DATA_BLOCK "pressure"   // DB71
{ S7_Optimized_Access := 'TRUE' }
VERSION : 0.1
// stored: AutoNumber true, DBAccessibleFromOPCUA true, IsOnlyStoredInLoadMemory false, IsRetainMemResEnabled false, IsWriteProtectedInAS false, MemoryReserve 100
   VAR RETAIN
      "A" : Struct
         "pressure at 20mA" : Real := 160.0;
         "Maximum Pressure user" : Real := 10.0;
         "maximum pressure Admin" : Real := 10.0;
         "minimum Pressure" : Real := 1.5;
      END_STRUCT;
      "B" : Struct
         "pressure at 20mA" : Real := 160.0;
         "Maximum Pressure user" : Real := 10.0;
         "maximum pressure Admin" : Real := 10.0;
         "minimum Pressure" : Real := 1.5;
      END_STRUCT;
   END_VAR
   VAR
      "Control A" : Struct
         "Over pressure occured" : Bool := FALSE;
         "under pressure Occured" : Bool := FALSE;
      END_STRUCT;
      "Control B" : Struct
         "Over pressure occured" : Bool := FALSE;
         "under pressure Occured" : Bool := FALSE;
      END_STRUCT;
      "pump A Inlet" : Real := 1.50463;
      "pump B Inlet" : Real := 1.545139;
      "pump A Outlet" : Real := 0.1808449;
      "pump B Outlet" : Real := 0.1139323;
      "Vessel A1 mbar" : DInt := 0;
      "Vessel A2 mbar" : DInt := 0;
      "Vessel B2 mbar" : DInt := 0;
      "Vessel B1 mbar" : DInt := 0;
   END_VAR
   VAR RETAIN
      "Over pressure Delay time user" : DInt := 1000;
      "over pressure delay time admin" : DInt := 10000;
      "under pressure delay time" : DInt := 1000;
      "Vaccum  sensor range" : Struct
         A1mbar : DInt := 9000;
         A2mbar : DInt := 9000;
         B1mbar : DInt := 9000;
         B2mbar : DInt := 9000;
         A1bar : Real := 9.0;
         A2bar : Real := 9.0;
         B1bar : Real := 9.0;
         B2bar : Real := 0.0;
      END_STRUCT;
   END_VAR
   VAR
      "vessel A1 bar" : Real := 0.0;
      "vessel A2 bar" : Real := 0.0;
      "vessel B1 bar" : Real := 0.0;
      "vessel B2 bar" : Real := 0.0;
      Misc : Struct
         "Pump A normx valueIN" : Real := 0.009403936;
         "Pump B normx valueIN" : Real := 0.009657118;
         "Pump A Scalx valueIN" : Real := 1.50463;
         "Pump B Scalx valueIN" : Real := 1.545139;
         "Pump A normx valueOUT" : Real := 0.007233796;
         "Pump B normx valueOUT" : Real := 0.004557292;
         "Pump A Scalx valueOUT" : Real := 0.1808449;
         "Pump B Scalx valueOUT" : Real := 0.1139323;
         "normx Tank A1" : Real := 0.0;
         "normx Tank A2" : Real := 0.0;
         "normx Tank B1" : Real := 0.0;
         "normx Tank B2" : Real := 0.0;
         "scalx Tank A1" : Real := 0.0;
         "scalx Tank A2" : Real := 0.0;
         "scalx Tank B1" : Real := 0.0;
         "scalx Tank B2" : Real := 0.0;
      END_STRUCT;
      "Control Vessel A1" : Struct
         "under pressure" : Bool := FALSE;
         "Over pressure open release valve" : Bool := FALSE;
      END_STRUCT;
      "Control Vessel A2" : Struct
         "under pressure" : Bool := FALSE;
         "Over pressure open release valve" : Bool := FALSE;
      END_STRUCT;
      "Control Vessel B1" : Struct
         "under pressure" : Bool := FALSE;
         "Over pressure open release valve" : Bool := FALSE;
      END_STRUCT;
      "Control Vessel B2" : Struct
         "under pressure" : Bool := FALSE;
         "Over pressure open release valve" : Bool := FALSE;
      END_STRUCT;
   END_VAR
   VAR RETAIN
      A_Outlet : Struct
         "pressure at 20mA" : Real := 25.0;
         "Maximum Pressure user" : Real := 20.0;
         "maximum pressure Admin" : Real := 20.0;
         "minimum Pressure" : Real := 1.0;
      END_STRUCT;
      B_Outlet : Struct
         "pressure at 20mA" : Real := 25.0;
         "Maximum Pressure user" : Real := 20.0;
         "maximum pressure Admin" : Real := 20.0;
         "minimum Pressure" : Real := 1.0;
      END_STRUCT;
   END_VAR
   VAR
      "Control A_Outlet" : Struct
         "Over pressure occured" : Bool := FALSE;
         "under pressure Occured" : Bool := FALSE;
      END_STRUCT;
      "Control B_Outlet" : Struct
         "Over pressure occured" : Bool := FALSE;
         "under pressure Occured" : Bool := FALSE;
      END_STRUCT;
   END_VAR
   VAR RETAIN
      Outlet_PT_ENABLE : Bool := TRUE;
   END_VAR
BEGIN
END_DATA_BLOCK

DATA_BLOCK "vessel"   // DB75
{ S7_Optimized_Access := 'TRUE' }
VERSION : 0.1
// stored: AutoNumber true, DBAccessibleFromOPCUA true, IsOnlyStoredInLoadMemory false, IsRetainMemResEnabled false, IsWriteProtectedInAS false, MemoryReserve 100
   VAR RETAIN
      "Duration pressure equalization" : Struct
         "A" : Int := 10;
         "B" : Int := 10;
      END_STRUCT;
      "amibient pressure" : Int := 900;
      "hysteresis ambient pressure" : Int := 50;
      "working pressure" : Struct
         "A" : Real := 3.0;
         "A+" : Real;
         "A-" : Real;
         "B" : Real := 3.0;
         "B+" : Real;
         "B-" : Real;
      END_STRUCT;
      "working pressure hysteresis" : Struct
         "A" : Real;
         "B" : Real;
      END_STRUCT;
   END_VAR
   VAR
      "Vaccum sensor selection" : Struct
         "selection A" : Int;
         "selection B" : Int;
         "A selected" : Bool;
         "B selected" : Bool;
         "A or B selected" : Bool;
      END_STRUCT;
      "Evacuation set Vaccum" : Struct
         A1 : Int;
         A2 : Int;
         B1 : Int;
         B2 : Int;
      END_STRUCT;
      "Evacuation Real vaccum" : Struct
         A1 : Int;
         A2 : Int;
         B1 : Int;
         B2 : Int;
      END_STRUCT;
      "Evacuation Time set" : Struct
         A1 : Int;
         A2 : Int;
         B1 : Int;
         B2 : Int;
      END_STRUCT;
      "Evacuation Time Real" : Struct
         A1 : Int;
         A2 : Int;
         B1 : Int;
         B2 : Int;
      END_STRUCT;
   END_VAR
   VAR RETAIN
      "preparation status" : Struct
         A1 : Int;
         A2 : Int;
         B1 : Int;
         B2 : Int;
      END_STRUCT;
      "monitor status" : Struct
         A1 : Int;
         A2 : Int;
         B1 : Int;
         B2 : Int;
      END_STRUCT;
      "Activate vessel" : Struct
         A1 : Bool;
         A2 : Bool;
         B1 : Bool;
         B2 : Bool;
      END_STRUCT;
   END_VAR
   VAR
      "A status" : Int;
      "B status" : Int;
   END_VAR
BEGIN
END_DATA_BLOCK

DATA_BLOCK "vessel_1"   // DB81
{ S7_Optimized_Access := 'TRUE' }
VERSION : 0.1
// stored: AutoNumber true, DBAccessibleFromOPCUA true, IsOnlyStoredInLoadMemory false, IsRetainMemResEnabled false, IsWriteProtectedInAS false, MemoryReserve 100
   VAR RETAIN
      "Duration pressure equalization" : Struct
         "A" : Int;
         "B" : Int;
      END_STRUCT;
      "amibient pressure" : Int;
      "hysteresis ambient pressure" : Int;
      "working pressure" : Struct
         "A" : Real;
         "A+" : Real;
         "A-" : Real;
         "B" : Real;
         "B+" : Real;
         "B-" : Real;
      END_STRUCT;
      "working pressure hysteresis" : Struct
         "A" : Real;
         "B" : Real;
      END_STRUCT;
   END_VAR
   VAR
      "Vaccum sensor selection" : Struct
         "selection A" : Int;
         "selection B" : Int;
         "A selected" : Bool;
         "B selected" : Bool;
         "A or B selected" : Bool;
      END_STRUCT;
      "Ready status" : Struct
         A1 : Int;
         A2 : Int;
         B1 : Int;
      END_STRUCT;
      "Evacuation set Vaccum" : Struct
         A1 : Int;
         A2 : Int;
         B1 : Int;
      END_STRUCT;
      "Evacuation Real vaccum" : Struct
         A1 : Int;
         A2 : Int;
         B1 : Int;
      END_STRUCT;
      "Evacuation Time set" : Struct
         A1 : Int;
         A2 : Int;
         B1 : Int;
      END_STRUCT;
      "Evacuation Time Real" : Struct
         A1 : Int;
         A2 : Int;
         B1 : Int;
      END_STRUCT;
   END_VAR
   VAR RETAIN
      "Active vessel" : Struct
         A1 : Bool;
         A2 : Bool;
         "A" : Bool;
         B1 : Bool;
      END_STRUCT;
      "preparation status" : Struct
         A1 : Int;
         A2 : Int;
         B1 : Int;
      END_STRUCT;
      "monitor status" : Struct
         "A" : Int;
         "B" : Int;
         C : Int;
      END_STRUCT;
      "Activate vessel" : Struct
         A1 : Bool;
         A2 : Bool;
         B1 : Bool;
      END_STRUCT;
   END_VAR
   VAR
      Ready : Struct
         A1 : Bool;
         A2 : Bool;
         B1 : Bool;
      END_STRUCT;
      "Activate vessel HMI" : Struct
         A1 : Bool;
         A2 : Bool;
         B1 : Bool;
      END_STRUCT;
      "DeActivate vessel HMI" : Struct
         A1 : Bool;
         A2 : Bool;
         B1 : Bool;
      END_STRUCT;
   END_VAR
BEGIN
END_DATA_BLOCK

DATA_BLOCK "Alarm_DB"   // DB36
{ S7_Optimized_Access := 'FALSE' }
VERSION : 0.1
// stored: AutoNumber true, DBAccessibleFromOPCUA true, IsOnlyStoredInLoadMemory false, IsWriteProtectedInAS false
   VAR
      input : Struct
         alarm : Array[0..95] of Bool;   // Connect the alarm inputs according to the alarm list
         ack : Array[0..95] of Bool;
      END_STRUCT;
      output : Struct
         alarm_reg : Array[0..95] of Bool;
      END_STRUCT;
      i : Int;
      alarmhmi : Bool;
      alarmRegister1 : Word;
      alarmRegister2 : Word;
      alarmRegister3 : Word;
      alarmRegister4 : Word;
      alarmRegister5 : Word;
      reset : Array[0..95] of Bool;
   END_VAR
BEGIN
   // input.alarm[0] : reg1 bit 8
   // input.alarm[1] : reg1 bit 9
   // input.alarm[2] : reg1 bit 10
   // input.alarm[3] : reg1 bit 11
   // input.alarm[4] : reg1 bit 12
   // input.alarm[5] : reg1 bit 13
   // input.alarm[6] : reg1 bit 14
   // input.alarm[7] : reg1 bit 15
   // input.alarm[8] : reg1 bit 0
   // input.alarm[9] : reg1 bit 1
   // input.alarm[10] : reg1 bit 2
   // input.alarm[11] : reg1 bit 3
   // input.alarm[12] : reg1 bit 4
   // input.alarm[13] : reg1 bit 5
   // input.alarm[14] : reg1 bit 6
   // input.alarm[15] : reg1 bit 0
   // input.alarm[16] : reg2 bit 8
   // input.alarm[17] : reg2 bit 9
   // input.alarm[18] : reg2 bit 10
   // input.alarm[19] : reg2 bit 11
   // input.alarm[20] : reg2 bit 12
   // input.alarm[21] : reg2 bit 13
   // input.alarm[22] : reg2 bit 14
   // input.alarm[23] : reg2 bit 15
   // input.alarm[24] : reg2 bit 7
   // input.alarm[25] : reg2 bit 6
   // input.alarm[26] : reg2 bit 5
   // input.alarm[27] : reg2 bit 4
   // input.alarm[28] : reg2 bit 3
   // input.alarm[29] : reg2 bit 2
   // input.alarm[30] : reg2 bit 1
   // input.alarm[31] : reg2 bit 0
   // input.alarm[32] : reg3 bit 8
   // input.alarm[33] : reg3 bit 9
   // input.alarm[34] : reg3 bit 10
   // input.alarm[35] : reg3 bit 11
   // input.alarm[36] : reg3 bit 12
   // input.alarm[37] : reg3 bit 13
   // input.alarm[38] : reg3 bit 14
   // input.alarm[39] : reg3 bit 15
   // input.alarm[40] : reg3 bit 7
   // input.alarm[41] : reg3 bit 6
   // input.alarm[42] : reg3 bit 5
   // input.alarm[43] : reg3 bit 4
   // input.alarm[44] : reg3 bit 3
   // input.alarm[45] : reg3 bit 2
   // input.alarm[46] : reg3 bit 1
   // input.alarm[47] : reg3 bit 0
   // input.alarm[48] : reg4 bit 8
   // input.alarm[49] : reg4 bit 9
   // input.alarm[50] : reg4 bit 10
   // input.alarm[51] : reg4 bit 11
   // input.alarm[52] : reg4 bit 12
   // input.alarm[53] : reg4 bit 13
   // input.alarm[54] : reg4 bit 14
   // input.alarm[55] : reg4 bit 15
   // input.alarm[56] : reg4 bit 7
   // input.alarm[57] : reg4 bit 6
   // input.alarm[58] : reg4 bit 5
   // input.alarm[59] : reg4 bit 4
   // input.alarm[60] : reg4 bit 3
   // input.alarm[61] : reg4 bit 2
   // input.alarm[62] : reg4 bit 1
   // input.alarm[63] : reg4 bit 0
   // input.alarm[64] : reg5 bit 8
   // input.alarm[65] : reg5 bit 9
   // input.alarm[66] : reg5 bit 10
   // input.alarm[67] : reg5 bit 11
   // input.alarm[68] : reg5 bit 12
   // input.alarm[69] : reg5 bit 13
   // input.alarm[70] : reg5 bit 14
   // input.alarm[71] : reg5 bit 15
   // input.alarm[72] : reg5 bit 7
   // input.alarm[73] : reg5 bit 6
   // input.alarm[74] : reg5 bit 5
   // input.alarm[75] : reg5 bit 4
   // input.alarm[76] : reg5 bit 3
   // input.alarm[77] : reg5 bit 2
   // input.alarm[78] : reg5 bit 1
   // input.alarm[79] : reg5 bit 0
END_DATA_BLOCK

DATA_BLOCK "Heater settings"   // DB138
{ S7_Optimized_Access := 'TRUE' }
VERSION : 0.1
// stored: AutoNumber true, DBAccessibleFromOPCUA true, IsOnlyStoredInLoadMemory false, IsRetainMemResEnabled false, IsWriteProtectedInAS false, MemoryReserve 100
   VAR RETAIN
      "Heater 1" : Struct
         "set temperature" : Real;
         "preshutdown temperature" : Real;
         "Limit under temparature" : Real;
         "Limit Over temperature" : Real;
         "Heating adjustment hysteresis" : Real;
         "Minimum ON time" : Real;
         "Minimum Off time" : Real;
      END_STRUCT;
      "Heater 2" : Struct
         "set temperature" : Real;
         "preshutdown temperature" : Real;
         "Limit under temparature" : Real;
         "Limit Over temperature" : Real;
         "Heating adjustment hysteresis" : Real;
         "Minimum ON time" : Real;
         "Minimum Off time" : Real;
      END_STRUCT;
      "Heater 3" : Struct
         "set temperature" : Real;
         "preshutdown temperature" : Real;
         "Limit under temparature" : Real;
         "Limit Over temperature" : Real;
         "Heating adjustment hysteresis" : Real;
         "Minimum ON time" : Real;
         "Minimum Off time" : Real;
      END_STRUCT;
      "Heater 4" : Struct
         "set temperature" : Real;
         "preshutdown temperature" : Real;
         "Limit under temparature" : Real;
         "Limit Over temperature" : Real;
         "Heating adjustment hysteresis" : Real;
         "Minimum ON time" : Real;
         "Minimum Off time" : Real;
      END_STRUCT;
      "heater EN 1" : Bool;
      "heater EN 2" : Bool;
      "heater EN 3" : Bool;
      "heater EN 4" : Bool;
   END_VAR
BEGIN
END_DATA_BLOCK

DATA_BLOCK "Heatercontrol"   // DB140
{ S7_Optimized_Access := 'TRUE' }
VERSION : 0.1
// stored: AutoNumber true, DBAccessibleFromOPCUA true, IsOnlyStoredInLoadMemory false, IsRetainMemResEnabled false, IsWriteProtectedInAS false, MemoryReserve 100
   VAR RETAIN
      ON : Struct
         heater1 : Bool;
         heater2 : Bool;
         heater3 : Bool;
         heater4 : Bool;
      END_STRUCT;
      "heater ON HMI" : Bool;
   END_VAR
   VAR
      "Show heater Button" : Bool;
   END_VAR
BEGIN
END_DATA_BLOCK

DATA_BLOCK "heater status"   // DB141
{ S7_Optimized_Access := 'TRUE' }
VERSION : 0.1
// stored: AutoNumber true, DBAccessibleFromOPCUA true, IsOnlyStoredInLoadMemory false, IsRetainMemResEnabled false, IsWriteProtectedInAS false, MemoryReserve 100
   VAR
      temperature : Struct
         heater1 : Real;
         heater2 : Real;
         heater3 : Real;
         heater4 : Real;
      END_STRUCT;
   END_VAR
   VAR RETAIN
      "p100 connection okay" : Struct
         heater1 : Bool;
         heater2 : Bool;
         heater3 : Bool;
         heater4 : Bool;
      END_STRUCT;
   END_VAR
   VAR
      "Limit under temperature" : Struct
         heater1 : Bool;
         heater2 : Bool;
         heater3 : Bool;
         heater4 : Bool;
      END_STRUCT;
      "Limit Over temperature" : Struct
         heater1 : Bool;
         heater2 : Bool;
         heater3 : Bool;
         heater4 : Bool;
      END_STRUCT;
      "Dispensing Stop under temperature heater" { ExternalAccessible := 'False'; ExternalVisible := 'False'; ExternalWritable := 'False'} : Array[1..4] of Bool;
      "Critical Fault Stop Dispense Temperature NOK" : Bool;
      heater_nok : Bool;
   END_VAR
BEGIN
END_DATA_BLOCK

DATA_BLOCK "selection_machie_db"   // DB18
{ S7_Optimized_Access := 'TRUE' }
VERSION : 0.1
// stored: AutoNumber true, DBAccessibleFromOPCUA true, IsOnlyStoredInLoadMemory false, IsRetainMemResEnabled false, IsWriteProtectedInAS false, MemoryReserve 100
   VAR
      "1k_2k" : Bool;
   END_VAR
BEGIN
END_DATA_BLOCK

ORGANIZATION_BLOCK "Main"   // OB1, LAD, ProgramCycle
TITLE = "Main Program Sweep (Cycle)"
{ S7_Optimized_Access := 'TRUE' }
VERSION : 0.1
// stored: AutoNumber true, IsIECCheckEnabled false, SetENOAutomatically false
   VAR_INPUT
      Initial_Call : Bool;   // Initial call of this OB
      Remanence : Bool;   // =True, if remanent data are available
   END_VAR
   VAR_TEMP
      temp1 : Bool;
      temp2 : Bool;
      temp3 : Bool;
      temp4 : Bool;
   END_VAR
   VAR_TEMP   // added for the SCL form of the ladder/FBD networks
      _w1 : Bool;
      _w2 : Bool;
      _w3 : Bool;
      _w4 : Bool;
      _w5 : Bool;
      _w6 : Bool;
      _w7 : Bool;
      _w8 : Bool;
      _w9 : Bool;
      _w10 : Bool;
      _w11 : Bool;
      _w12 : Bool;
      _w13 : Bool;
      _w14 : Bool;
      _w15 : Bool;
      _w16 : Bool;
   END_VAR
BEGIN

REGION Network 1: SFC1
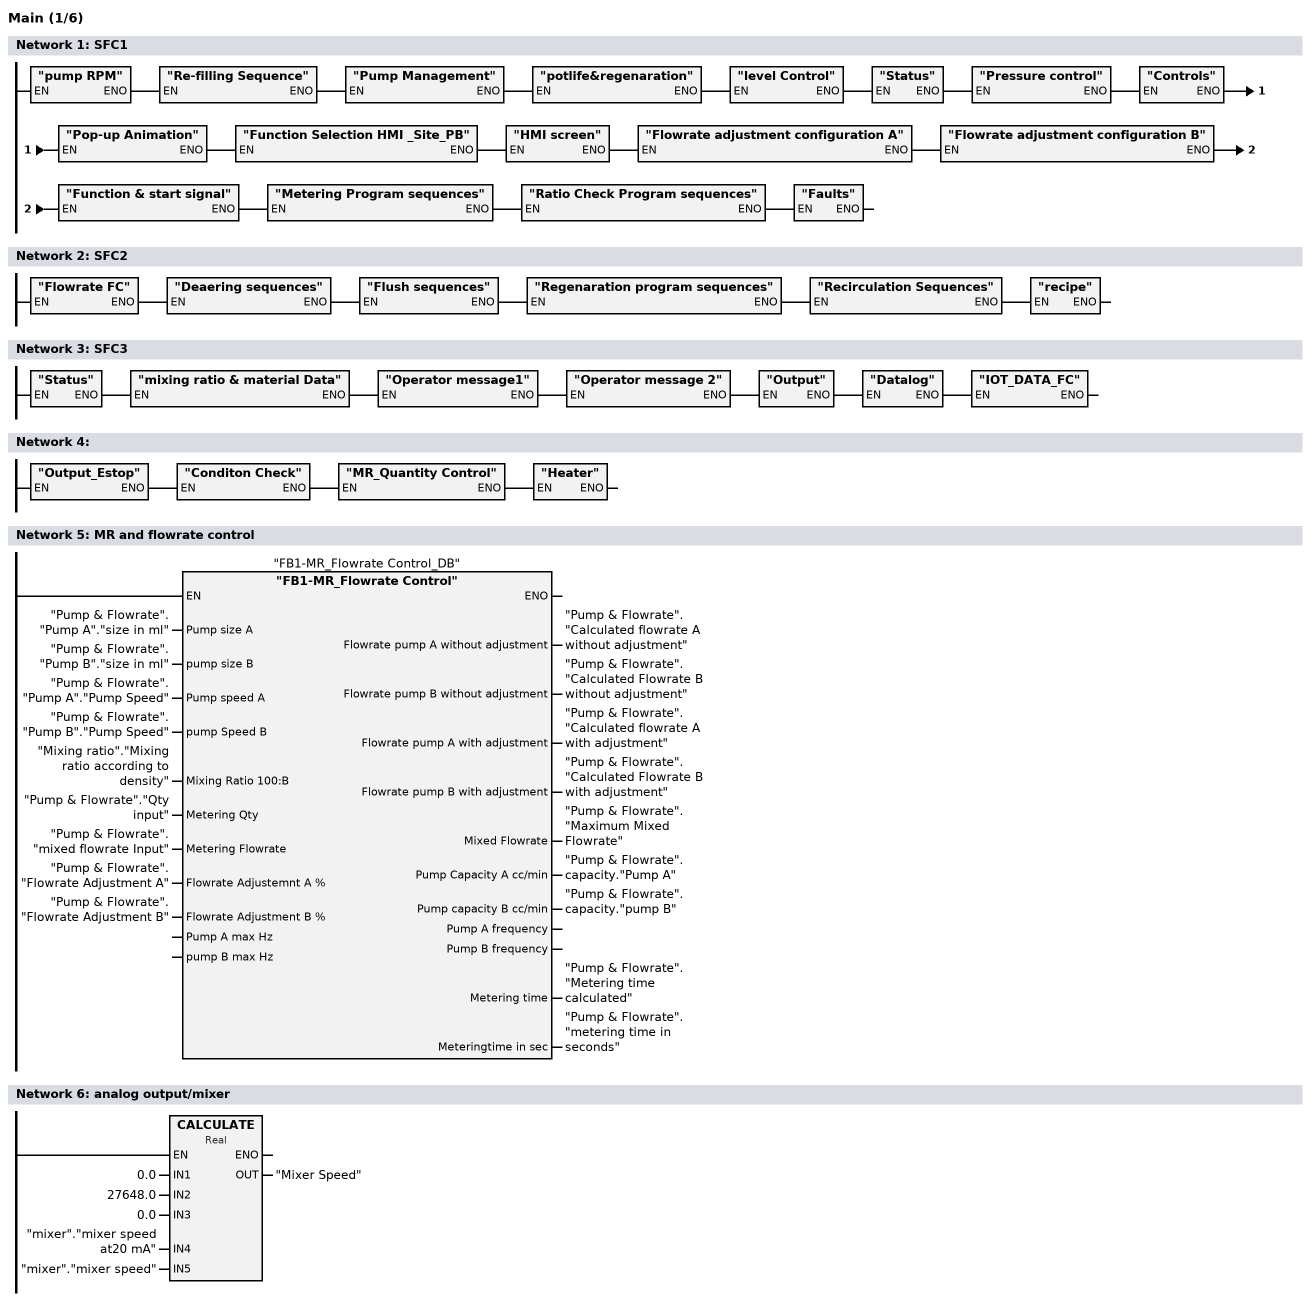
   RUNG wire#powerrail
      "pump RPM"()
      "Re-filling Sequence"()
      "Pump Management"()
      "potlife&regenaration"()
      "level Control"()
      "Status"()
      "Pressure control"()
      "Controls"()
      "Pop-up Animation"()
      "Function Selection HMI _Site_PB"()
      "HMI screen"()
      "Flowrate adjustment configuration A"()
      "Flowrate adjustment configuration B"()
      "Function & start signal"()
      "Metering Program sequences"()
      "Ratio Check Program sequences"()
      "Faults"()
   END_RUNG
   // the same network as SCL:
   "pump RPM"(ENO => #_w1);
   "Re-filling Sequence"(EN := #_w1, ENO => #_w2);
   "Pump Management"(EN := #_w2, ENO => #_w3);
   "potlife&regenaration"(EN := #_w3, ENO => #_w4);
   "level Control"(EN := #_w4, ENO => #_w5);
   "Status"(EN := #_w5, ENO => #_w6);
   "Pressure control"(EN := #_w6, ENO => #_w7);
   "Controls"(EN := #_w7, ENO => #_w8);
   "Pop-up Animation"(EN := #_w8, ENO => #_w9);
   "Function Selection HMI _Site_PB"(EN := #_w9, ENO => #_w10);
   "HMI screen"(EN := #_w10, ENO => #_w11);
   "Flowrate adjustment configuration A"(EN := #_w11, ENO => #_w12);
   "Flowrate adjustment configuration B"(EN := #_w12, ENO => #_w13);
   "Function & start signal"(EN := #_w13, ENO => #_w14);
   "Metering Program sequences"(EN := #_w14, ENO => #_w15);
   "Ratio Check Program sequences"(EN := #_w15, ENO => #_w16);
   IF #_w16 THEN "Faults"(); END_IF;
END_REGION

REGION Network 2: SFC2
   RUNG wire#powerrail
      "Flowrate FC"()
      "Deaering sequences"()
      "Flush sequences"()
      "Regenaration program sequences"()
      "Recirculation Sequences"()
      "recipe"()
   END_RUNG
   // the same network as SCL:
   "Flowrate FC"(ENO => #_w1);
   "Deaering sequences"(EN := #_w1, ENO => #_w2);
   "Flush sequences"(EN := #_w2, ENO => #_w3);
   "Regenaration program sequences"(EN := #_w3, ENO => #_w4);
   "Recirculation Sequences"(EN := #_w4, ENO => #_w5);
   IF #_w5 THEN "recipe"(); END_IF;
END_REGION

REGION Network 3: SFC3
   RUNG wire#powerrail
      "Status"()
      "mixing ratio & material Data"()
      "Operator message1"()
      "Operator message 2"()
      "Output"()
      "Datalog"()
      "IOT_DATA_FC"()
   END_RUNG
   // the same network as SCL:
   "Status"(ENO => #_w1);
   "mixing ratio & material Data"(EN := #_w1, ENO => #_w2);
   "Operator message1"(EN := #_w2, ENO => #_w3);
   "Operator message 2"(EN := #_w3, ENO => #_w4);
   "Output"(EN := #_w4, ENO => #_w5);
   "Datalog"(EN := #_w5, ENO => #_w6);
   IF #_w6 THEN "IOT_DATA_FC"(); END_IF;
END_REGION

REGION Network 4
   RUNG wire#powerrail
      "Output_Estop"()
      "Conditon Check"()
      "MR_Quantity Control"()
      "Heater"()
   END_RUNG
   // the same network as SCL:
   "Output_Estop"(ENO => #_w1);
   "Conditon Check"(EN := #_w1, ENO => #_w2);
   "MR_Quantity Control"(EN := #_w2, ENO => #_w3);
   IF #_w3 THEN "Heater"(); END_IF;
END_REGION

REGION Network 5: MR and flowrate control
   "FB1-MR_Flowrate Control_DB"("Pump size A" := "Pump & Flowrate"."Pump A"."size in ml",   // "FB1-MR_Flowrate Control"
                           "pump size B" := "Pump & Flowrate"."Pump B"."size in ml",
                           "Pump speed A" := "Pump & Flowrate"."Pump A"."Pump Speed",
                           "pump Speed B" := "Pump & Flowrate"."Pump B"."Pump Speed",
                           "Mixing Ratio 100:B" := "Mixing ratio"."Mixing ratio according to density",
                           "Metering Qty" := "Pump & Flowrate"."Qty input",
                           "Metering Flowrate" := "Pump & Flowrate"."mixed flowrate Input",
                           "Flowrate Adjustemnt A %" := "Pump & Flowrate"."Flowrate Adjustment A",
                           "Flowrate Adjustment B %" := "Pump & Flowrate"."Flowrate Adjustment B",
                           "Flowrate pump A without adjustment" => "Pump & Flowrate"."Calculated flowrate A without adjustment",
                           "Flowrate pump B without adjustment" => "Pump & Flowrate"."Calculated Flowrate B without adjustment",
                           "Flowrate pump A with adjustment" => "Pump & Flowrate"."Calculated flowrate A with adjustment",
                           "Flowrate pump B with adjustment" => "Pump & Flowrate"."Calculated Flowrate B  with adjustment",
                           "Mixed Flowrate" => "Pump & Flowrate"."Maximum Mixed Flowrate",
                           "Pump Capacity A cc/min" => "Pump & Flowrate".capacity."Pump A",
                           "Pump capacity B cc/min" => "Pump & Flowrate".capacity."pump B",
                           "Metering time" => "Pump & Flowrate"."Metering time calculated",
                           "Meteringtime in sec" => "Pump & Flowrate"."metering time in seconds");
END_REGION

REGION Network 6: analog output/mixer
   RUNG wire#powerrail
      { S7_Templates := "SrcType := Real"; S7_Expression := "(IN2-IN1)*(IN5-IN3)/(IN4-IN3)+IN1" } Calculate(in1 := 0.0, in2 := 27648.0, in3 := 0.0, in4 := "mixer"."mixer speed at20 mA", in5 := "mixer"."mixer speed", out => "Mixer Speed")
   END_RUNG
   // the same network as SCL:
   "Mixer Speed" := (27648.0-0.0)*("mixer"."mixer speed"-0.0)/("mixer"."mixer speed at20 mA"-0.0)+0.0;
END_REGION

REGION Network 7: Pump A Analog output without PID
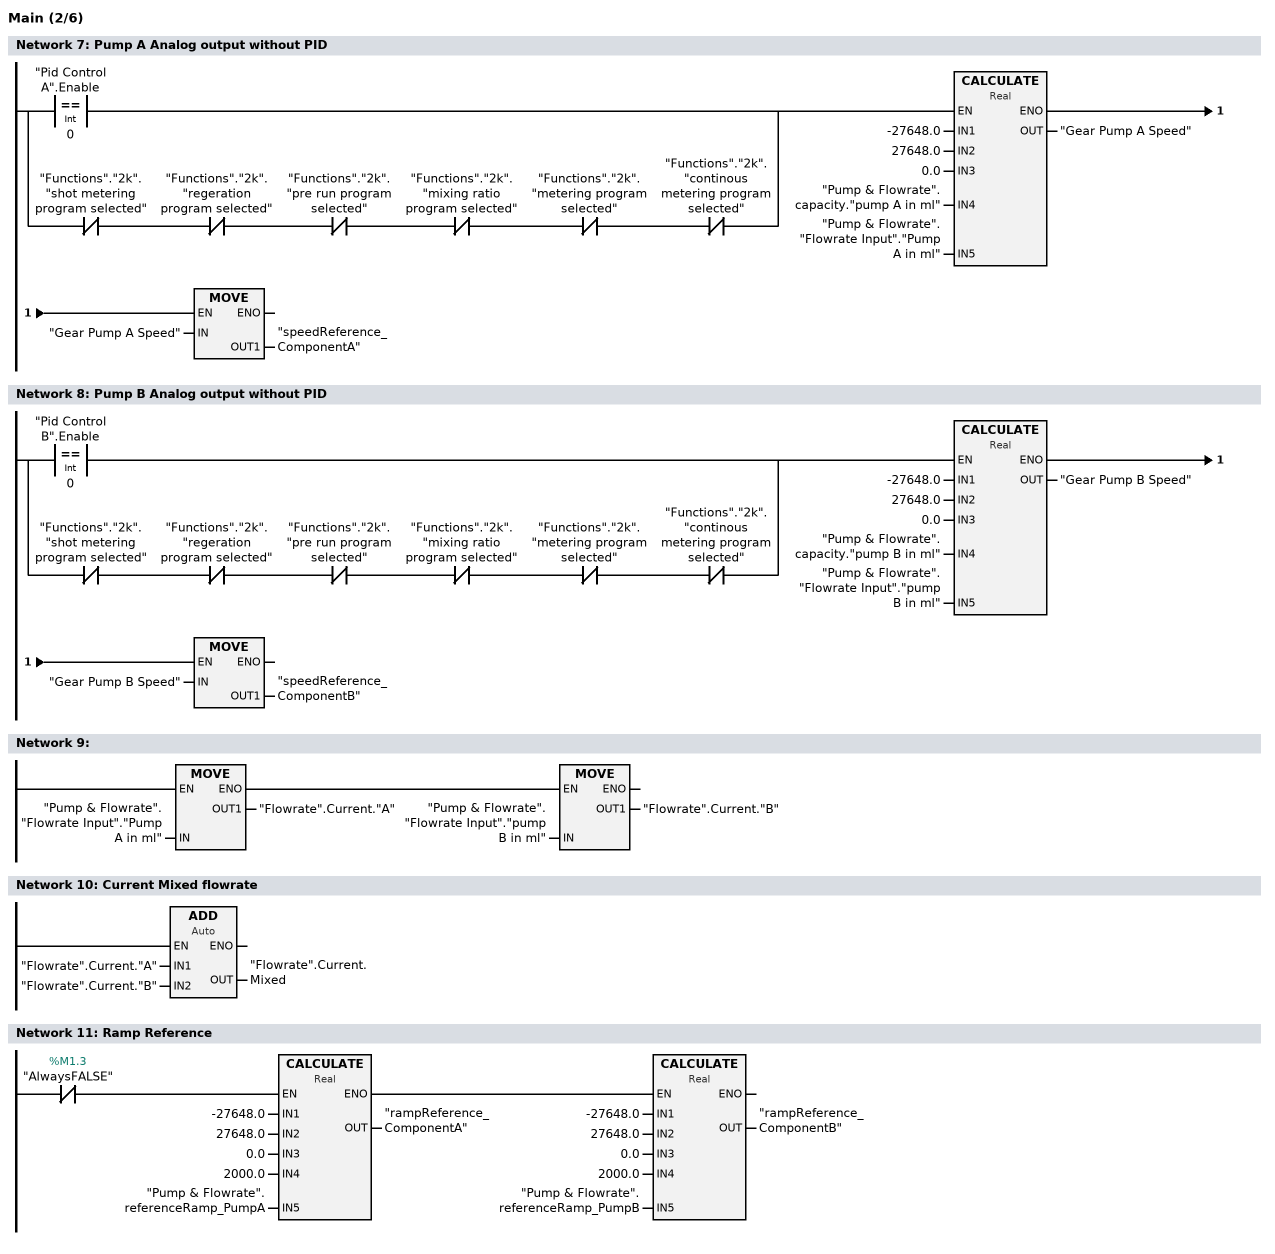
   RUNG wire#powerrail
      { S7_Templates := "SrcType := Int" } EQ_Contact(in1 := "Pid Control A".Enable, in2 := 0)
      wire#w1
      { S7_Templates := "SrcType := Real"; S7_Expression := "(IN2-IN1)*(IN5-IN3)/(IN4-IN3)+IN1" } Calculate(in1 := -27648.0, in2 := 27648.0, in3 := 0.0, in4 := "Pump & Flowrate".capacity."pump A in ml", in5 := "Pump & Flowrate"."Flowrate Input"."Pump A in ml", out => "Gear Pump A Speed")
      Move(in := "Gear Pump A Speed", out1 => "speedReference_ComponentA")
   END_RUNG
   RUNG wire#powerrail
      I_Contact( "Functions"."2k"."shot metering program selected" )
      I_Contact( "Functions"."2k"."regeration program selected" )
      I_Contact( "Functions"."2k"."pre run program selected" )
      I_Contact( "Functions"."2k"."mixing ratio program selected" )
      I_Contact( "Functions"."2k"."metering program selected" )
      I_Contact( "Functions"."2k"."continous metering program selected" )
   END_RUNG wire#w1
   // the same network as SCL:
   IF ("Pid Control A".Enable = 0) OR (NOT "Functions"."2k"."shot metering program selected" AND NOT "Functions"."2k"."regeration program selected" AND NOT "Functions"."2k"."pre run program selected" AND NOT "Functions"."2k"."mixing ratio program selected" AND NOT "Functions"."2k"."metering program selected" AND NOT "Functions"."2k"."continous metering program selected") THEN
       "Gear Pump A Speed" := (27648.0-(-27648.0))*("Pump & Flowrate"."Flowrate Input"."Pump A in ml"-0.0)/("Pump & Flowrate".capacity."pump A in ml"-0.0)+(-27648.0);
       "speedReference_ComponentA" := "Gear Pump A Speed";
   END_IF;
END_REGION

REGION Network 8: Pump B Analog output without PID
   RUNG wire#powerrail
      { S7_Templates := "SrcType := Int" } EQ_Contact(in1 := "Pid Control B".Enable, in2 := 0)
      wire#w1
      { S7_Templates := "SrcType := Real"; S7_Expression := "(IN2-IN1)*(IN5-IN3)/(IN4-IN3)+IN1" } Calculate(in1 := -27648.0, in2 := 27648.0, in3 := 0.0, in4 := "Pump & Flowrate".capacity."pump B in ml", in5 := "Pump & Flowrate"."Flowrate Input"."pump B in ml", out => "Gear Pump B Speed")
      Move(in := "Gear Pump B Speed", out1 => "speedReference_ComponentB")
   END_RUNG
   RUNG wire#powerrail
      I_Contact( "Functions"."2k"."shot metering program selected" )
      I_Contact( "Functions"."2k"."regeration program selected" )
      I_Contact( "Functions"."2k"."pre run program selected" )
      I_Contact( "Functions"."2k"."mixing ratio program selected" )
      I_Contact( "Functions"."2k"."metering program selected" )
      I_Contact( "Functions"."2k"."continous metering program selected" )
   END_RUNG wire#w1
   // the same network as SCL:
   IF ("Pid Control B".Enable = 0) OR (NOT "Functions"."2k"."shot metering program selected" AND NOT "Functions"."2k"."regeration program selected" AND NOT "Functions"."2k"."pre run program selected" AND NOT "Functions"."2k"."mixing ratio program selected" AND NOT "Functions"."2k"."metering program selected" AND NOT "Functions"."2k"."continous metering program selected") THEN
       "Gear Pump B Speed" := (27648.0-(-27648.0))*("Pump & Flowrate"."Flowrate Input"."pump B in ml"-0.0)/("Pump & Flowrate".capacity."pump B in ml"-0.0)+(-27648.0);
       "speedReference_ComponentB" := "Gear Pump B Speed";
   END_IF;
END_REGION

REGION Network 9
   RUNG wire#powerrail
      Move(in := "Pump & Flowrate"."Flowrate Input"."Pump A in ml", out1 => "Flowrate".Current."A")
      Move(in := "Pump & Flowrate"."Flowrate Input"."pump B in ml", out1 => "Flowrate".Current."B")
   END_RUNG
   // the same network as SCL:
   "Flowrate".Current."A" := "Pump & Flowrate"."Flowrate Input"."Pump A in ml";
   "Flowrate".Current."B" := "Pump & Flowrate"."Flowrate Input"."pump B in ml";
END_REGION

REGION Network 10: Current Mixed flowrate
   RUNG wire#powerrail
      Add(in1 := "Flowrate".Current."A", in2 := "Flowrate".Current."B", out => "Flowrate".Current.Mixed)
   END_RUNG
   // the same network as SCL:
   "Flowrate".Current.Mixed := "Flowrate".Current."A" + "Flowrate".Current."B";
END_REGION

REGION Network 11: Ramp Reference
   RUNG wire#powerrail
      I_Contact( "AlwaysFALSE" )
      { S7_Templates := "SrcType := Real"; S7_Expression := "ROUND((IN2-IN1)*(IN5-IN3)/(IN4-IN3)+IN1)" } Calculate(in1 := -27648.0, in2 := 27648.0, in3 := 0.0, in4 := 2000.0, in5 := "Pump & Flowrate".referenceRamp_PumpA, out => "rampReference_ComponentA")
      { S7_Templates := "SrcType := Real"; S7_Expression := "(IN2-IN1)*(IN5-IN3)/(IN4-IN3)+IN1" } Calculate(in1 := -27648.0, in2 := 27648.0, in3 := 0.0, in4 := 2000.0, in5 := "Pump & Flowrate".referenceRamp_PumpB, out => "rampReference_ComponentB")
   END_RUNG
   // the same network as SCL:
   IF NOT "AlwaysFALSE" THEN
       "rampReference_ComponentA" := ROUND((27648.0-(-27648.0))*("Pump & Flowrate".referenceRamp_PumpA-0.0)/(2000.0-0.0)+(-27648.0));
       "rampReference_ComponentB" := (27648.0-(-27648.0))*("Pump & Flowrate".referenceRamp_PumpB-0.0)/(2000.0-0.0)+(-27648.0);
   END_IF;
END_REGION

REGION Network 12: 2k Dosing running
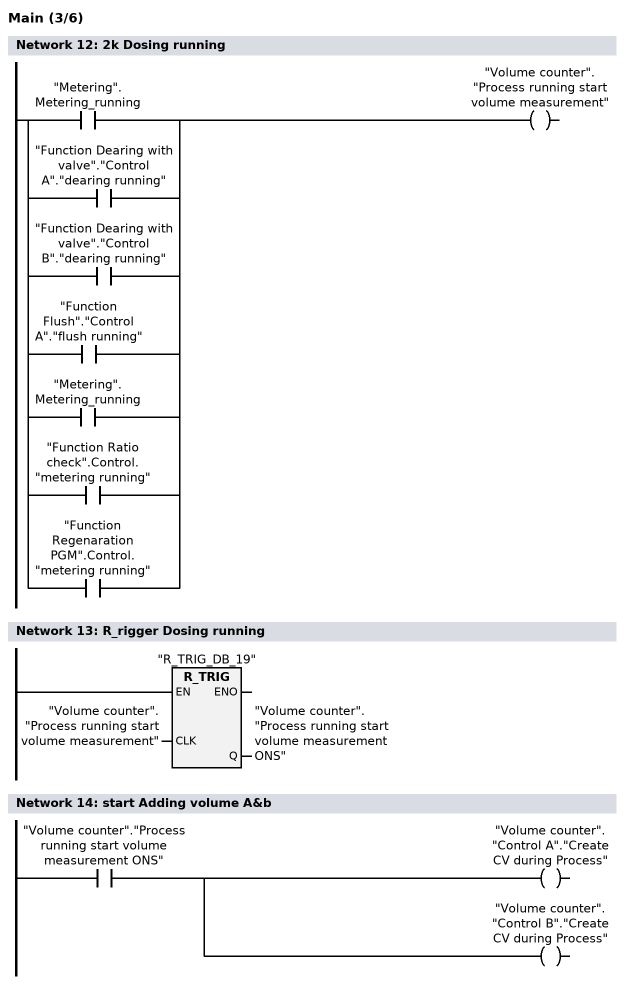
   RUNG wire#powerrail
      Contact( "Metering".Metering_running )
      wire#w1
      Coil( "Volume counter"."Process running start volume measurement" )
   END_RUNG
   RUNG wire#powerrail
      Contact( "Function Dearing with valve"."Control A"."dearing running" )
   END_RUNG wire#w1
   RUNG wire#powerrail
      Contact( "Function Dearing with valve"."Control B"."dearing running" )
   END_RUNG wire#w1
   RUNG wire#powerrail
      Contact( "Function Flush"."Control A"."flush running" )
   END_RUNG wire#w1
   RUNG wire#powerrail
      Contact( "Metering".Metering_running )
   END_RUNG wire#w1
   RUNG wire#powerrail
      Contact( "Function Ratio check".Control."metering running" )
   END_RUNG wire#w1
   RUNG wire#powerrail
      Contact( "Function Regenaration PGM".Control."metering running" )
   END_RUNG wire#w1
   // the same network as SCL:
   "Volume counter"."Process running start volume measurement" := "Metering".Metering_running OR "Function Dearing with valve"."Control A"."dearing running" OR "Function Dearing with valve"."Control B"."dearing running" OR "Function Flush"."Control A"."flush running" OR "Metering".Metering_running OR "Function Ratio check".Control."metering running" OR "Function Regenaration PGM".Control."metering running";
END_REGION

REGION Network 13: R_rigger Dosing running
   RUNG wire#powerrail
      "R_TRIG_DB_19".R_TRIG(CLK := "Volume counter"."Process running start volume measurement", Q => "Volume counter"."Process running start volume measurement ONS")
   END_RUNG
   // the same network as SCL:
   "R_TRIG_DB_19"(CLK := "Volume counter"."Process running start volume measurement",   // R_TRIG
                  Q => "Volume counter"."Process running start volume measurement ONS");
END_REGION

REGION Network 14: start Adding volume A&b
   RUNG wire#powerrail
      Contact( "Volume counter"."Process running start volume measurement ONS" )
      wire#w1
      Coil( "Volume counter"."Control A"."Create CV during Process" )
   END_RUNG
   RUNG wire#w1
      Coil( "Volume counter"."Control B"."Create CV during Process" )
   END_RUNG
   // the same network as SCL:
   "Volume counter"."Control A"."Create CV during Process" := "Volume counter"."Process running start volume measurement ONS";
   "Volume counter"."Control B"."Create CV during Process" := "Volume counter"."Process running start volume measurement ONS";
END_REGION

REGION Network 15: A volume During Operation
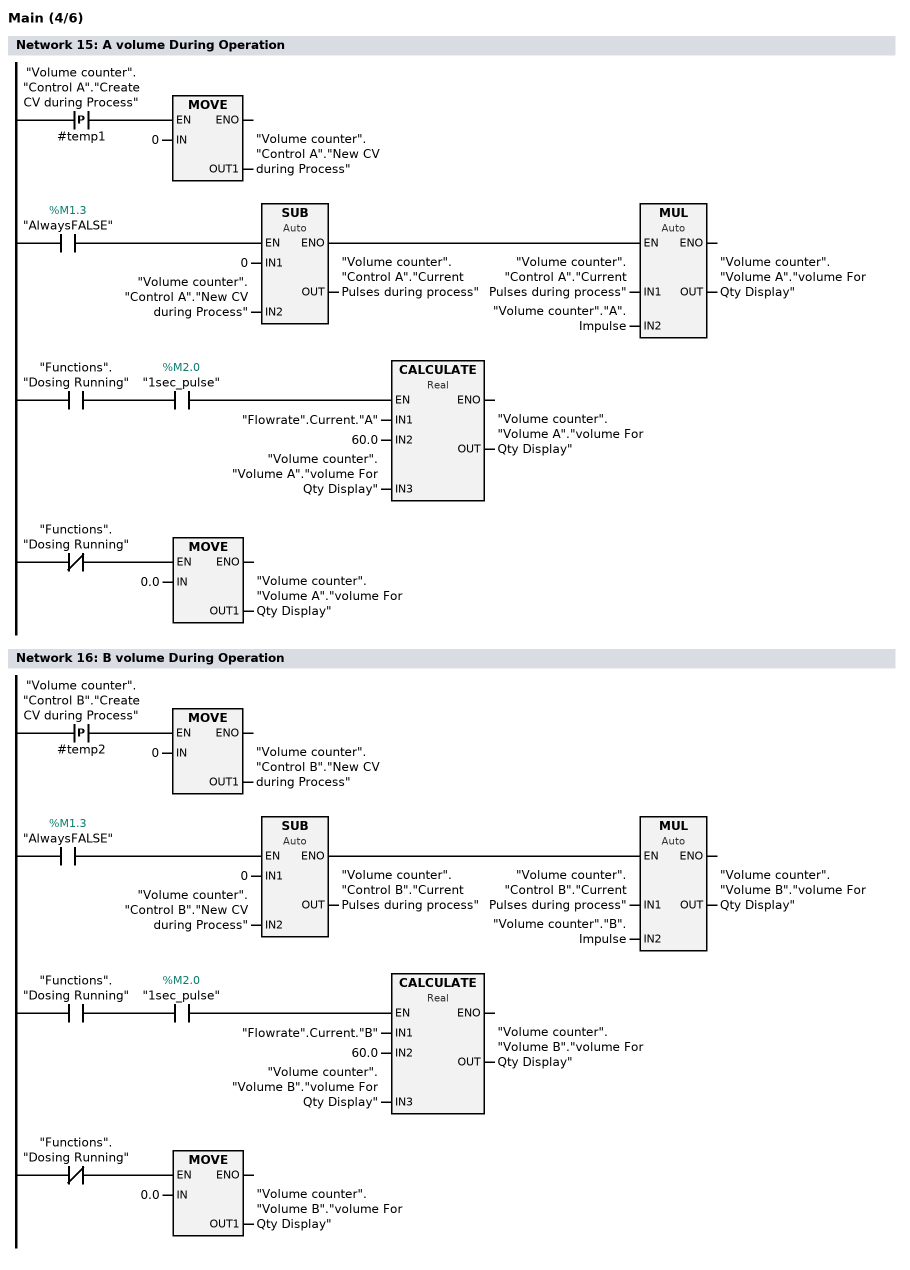
   RUNG wire#powerrail
      P_Contact(operand := "Volume counter"."Control A"."Create CV during Process", bit := #temp1)
      Move(in := 0, out1 => "Volume counter"."Control A"."New CV during Process")
   END_RUNG
   RUNG wire#powerrail
      Contact( "AlwaysFALSE" )
      Sub(in1 := 0, in2 := "Volume counter"."Control A"."New CV during Process", out => "Volume counter"."Control A"."Current Pulses during process")
      Mul(in1 := "Volume counter"."Control A"."Current Pulses during process", in2 := "Volume counter"."A".Impulse, out => "Volume counter"."Volume A"."volume For Qty Display")
   END_RUNG
   RUNG wire#powerrail
      Contact( "Functions"."Dosing Running" )
      Contact( "1sec_pulse" )
      { S7_Templates := "SrcType := Real"; S7_Expression := "(IN1/IN2)+IN3" } Calculate(in1 := "Flowrate".Current."A", in2 := 60.0, in3 := "Volume counter"."Volume A"."volume For Qty Display", out => "Volume counter"."Volume A"."volume For Qty Display")
   END_RUNG
   RUNG wire#powerrail
      I_Contact( "Functions"."Dosing Running" )
      Move(in := 0.0, out1 => "Volume counter"."Volume A"."volume For Qty Display")
   END_RUNG
   // the same network as SCL:
   #_w1 := "Volume counter"."Control A"."Create CV during Process" AND NOT #temp1;   // rising edge of "Volume counter"."Control A"."Create CV during Process"
   #temp1 := "Volume counter"."Control A"."Create CV during Process";
   IF #_w1 THEN "Volume counter"."Control A"."New CV during Process" := 0; END_IF;
   IF "AlwaysFALSE" THEN
       "Volume counter"."Control A"."Current Pulses during process" := 0 - "Volume counter"."Control A"."New CV during Process";
       "Volume counter"."Volume A"."volume For Qty Display" := "Volume counter"."Control A"."Current Pulses during process" * "Volume counter"."A".Impulse;
   END_IF;
   IF "Functions"."Dosing Running" AND "1sec_pulse" THEN
       "Volume counter"."Volume A"."volume For Qty Display" := ("Flowrate".Current."A"/60.0)+"Volume counter"."Volume A"."volume For Qty Display";
   END_IF;
   IF NOT "Functions"."Dosing Running" THEN
       "Volume counter"."Volume A"."volume For Qty Display" := 0.0;
   END_IF;
END_REGION

REGION Network 16: B volume During Operation
   RUNG wire#powerrail
      P_Contact(operand := "Volume counter"."Control B"."Create CV during Process", bit := #temp2)
      Move(in := 0, out1 => "Volume counter"."Control B"."New CV during Process")
   END_RUNG
   RUNG wire#powerrail
      Contact( "AlwaysFALSE" )
      Sub(in1 := 0, in2 := "Volume counter"."Control B"."New CV during Process", out => "Volume counter"."Control B"."Current Pulses during process")
      Mul(in1 := "Volume counter"."Control B"."Current Pulses during process", in2 := "Volume counter"."B".Impulse, out => "Volume counter"."Volume B"."volume For Qty Display")
   END_RUNG
   RUNG wire#powerrail
      Contact( "Functions"."Dosing Running" )
      Contact( "1sec_pulse" )
      { S7_Templates := "SrcType := Real"; S7_Expression := "(IN1/IN2)+IN3" } Calculate(in1 := "Flowrate".Current."B", in2 := 60.0, in3 := "Volume counter"."Volume B"."volume For Qty Display", out => "Volume counter"."Volume B"."volume For Qty Display")
   END_RUNG
   RUNG wire#powerrail
      I_Contact( "Functions"."Dosing Running" )
      Move(in := 0.0, out1 => "Volume counter"."Volume B"."volume For Qty Display")
   END_RUNG
   // the same network as SCL:
   #_w1 := "Volume counter"."Control B"."Create CV during Process" AND NOT #temp2;   // rising edge of "Volume counter"."Control B"."Create CV during Process"
   #temp2 := "Volume counter"."Control B"."Create CV during Process";
   IF #_w1 THEN "Volume counter"."Control B"."New CV during Process" := 0; END_IF;
   IF "AlwaysFALSE" THEN
       "Volume counter"."Control B"."Current Pulses during process" := 0 - "Volume counter"."Control B"."New CV during Process";
       "Volume counter"."Volume B"."volume For Qty Display" := "Volume counter"."Control B"."Current Pulses during process" * "Volume counter"."B".Impulse;
   END_IF;
   IF "Functions"."Dosing Running" AND "1sec_pulse" THEN
       "Volume counter"."Volume B"."volume For Qty Display" := ("Flowrate".Current."B"/60.0)+"Volume counter"."Volume B"."volume For Qty Display";
   END_IF;
   IF NOT "Functions"."Dosing Running" THEN
       "Volume counter"."Volume B"."volume For Qty Display" := 0.0;
   END_IF;
END_REGION

REGION Network 17: Mixed Volume During Operation
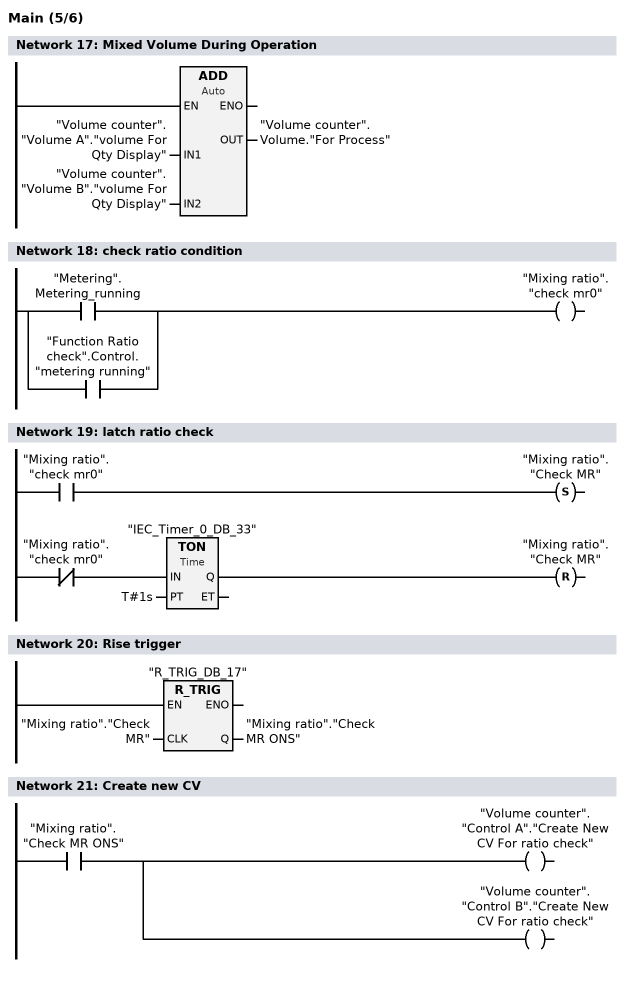
   RUNG wire#powerrail
      Add(in1 := "Volume counter"."Volume A"."volume For Qty Display", in2 := "Volume counter"."Volume B"."volume For Qty Display", out => "Volume counter".Volume."For Process")
   END_RUNG
   // the same network as SCL:
   "Volume counter".Volume."For Process" := "Volume counter"."Volume A"."volume For Qty Display" + "Volume counter"."Volume B"."volume For Qty Display";
END_REGION

REGION Network 18: check ratio condition
   RUNG wire#powerrail
      Contact( "Metering".Metering_running )
      wire#w1
      Coil( "Mixing ratio"."check mr0" )
   END_RUNG
   RUNG wire#powerrail
      Contact( "Function Ratio check".Control."metering running" )
   END_RUNG wire#w1
   // the same network as SCL:
   "Mixing ratio"."check mr0" := "Metering".Metering_running OR "Function Ratio check".Control."metering running";
END_REGION

REGION Network 19: latch ratio check
   RUNG wire#powerrail
      Contact( "Mixing ratio"."check mr0" )
      S_Coil( "Mixing ratio"."Check MR" )
   END_RUNG
   RUNG wire#powerrail
      I_Contact( "Mixing ratio"."check mr0" )
      { S7_Templates := "time_type := Time" } "IEC_Timer_0_DB_33".TON(pt := T#1s, et =>)
      R_Coil( "Mixing ratio"."Check MR" )
   END_RUNG
   // the same network as SCL:
   IF "Mixing ratio"."check mr0" THEN "Mixing ratio"."Check MR" := TRUE; END_IF;
   "IEC_Timer_0_DB_33".TON(IN := NOT "Mixing ratio"."check mr0", PT := T#1s);
   IF "IEC_Timer_0_DB_33".Q THEN "Mixing ratio"."Check MR" := FALSE; END_IF;
END_REGION

REGION Network 20: Rise trigger
   RUNG wire#powerrail
      "R_TRIG_DB_17".R_TRIG(CLK := "Mixing ratio"."Check MR", Q => "Mixing ratio"."Check MR ONS")
   END_RUNG
   // the same network as SCL:
   "R_TRIG_DB_17"(CLK := "Mixing ratio"."Check MR", Q => "Mixing ratio"."Check MR ONS");   // R_TRIG
END_REGION

REGION Network 21: Create new CV
   RUNG wire#powerrail
      Contact( "Mixing ratio"."Check MR ONS" )
      wire#w1
      Coil( "Volume counter"."Control A"."Create New CV For ratio check" )
   END_RUNG
   RUNG wire#w1
      Coil( "Volume counter"."Control B"."Create New CV For ratio check" )
   END_RUNG
   // the same network as SCL:
   "Volume counter"."Control A"."Create New CV For ratio check" := "Mixing ratio"."Check MR ONS";
   "Volume counter"."Control B"."Create New CV For ratio check" := "Mixing ratio"."Check MR ONS";
END_REGION

REGION Network 22: A volume During ratio check
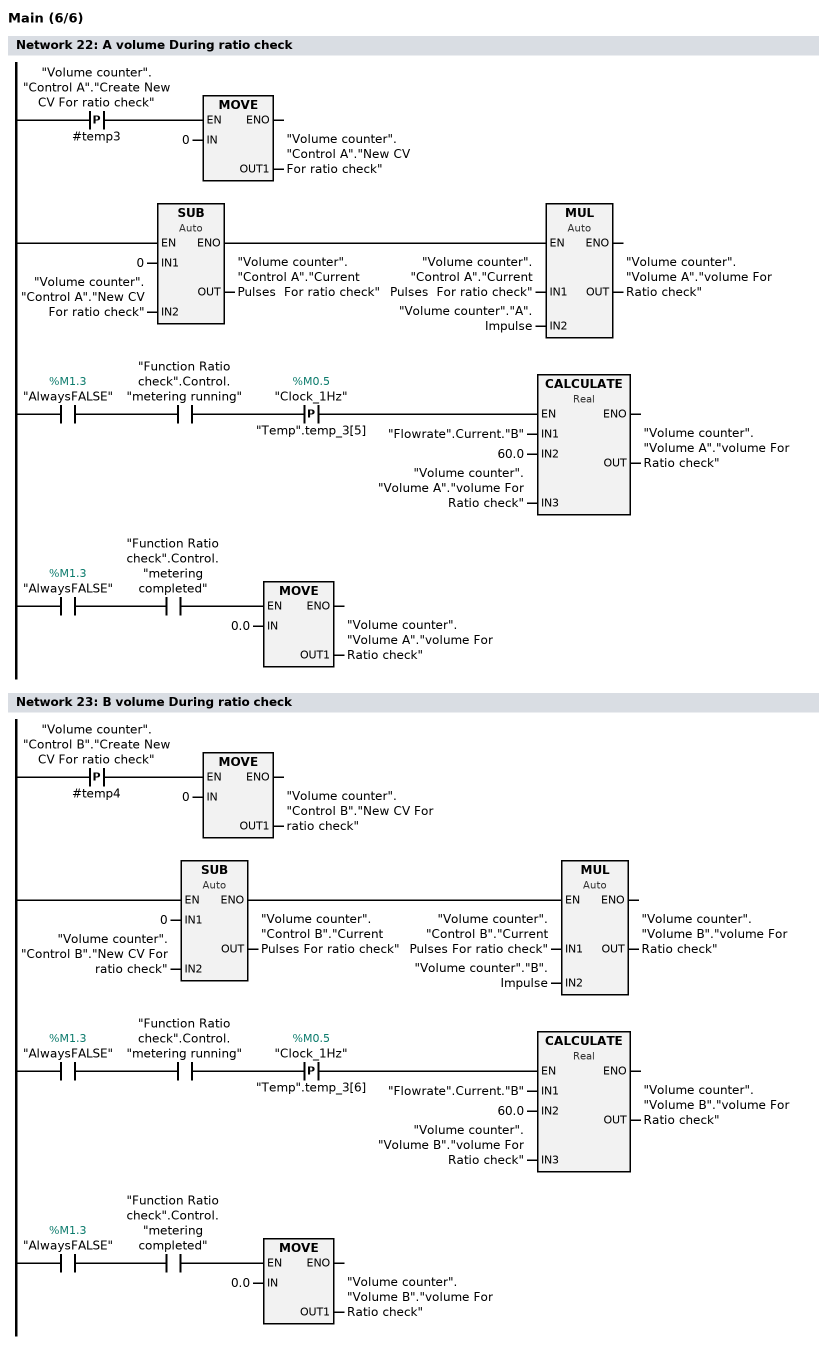
   RUNG wire#powerrail
      P_Contact(operand := "Volume counter"."Control A"."Create New CV For ratio check", bit := #temp3)
      Move(in := 0, out1 => "Volume counter"."Control A"."New CV  For ratio check")
   END_RUNG
   RUNG wire#powerrail
      Sub(in1 := 0, in2 := "Volume counter"."Control A"."New CV  For ratio check", out => "Volume counter"."Control A"."Current Pulses  For ratio check")
      Mul(in1 := "Volume counter"."Control A"."Current Pulses  For ratio check", in2 := "Volume counter"."A".Impulse, out => "Volume counter"."Volume A"."volume For Ratio check")
   END_RUNG
   RUNG wire#powerrail
      Contact( "AlwaysFALSE" )
      Contact( "Function Ratio check".Control."metering running" )
      P_Contact(operand := "Clock_1Hz", bit := "Temp".temp_3[5])
      { S7_Templates := "SrcType := Real"; S7_Expression := "(IN1/IN2)+IN3" } Calculate(in1 := "Flowrate".Current."B", in2 := 60.0, in3 := "Volume counter"."Volume A"."volume For Ratio check", out => "Volume counter"."Volume A"."volume For Ratio check")
   END_RUNG
   RUNG wire#powerrail
      Contact( "AlwaysFALSE" )
      Contact( "Function Ratio check".Control."metering completed" )
      Move(in := 0.0, out1 => "Volume counter"."Volume A"."volume For Ratio check")
   END_RUNG
   // the same network as SCL:
   #_w1 := "Volume counter"."Control A"."Create New CV For ratio check" AND NOT #temp3;   // rising edge of "Volume counter"."Control A"."Create New CV For ratio check"
   #temp3 := "Volume counter"."Control A"."Create New CV For ratio check";
   IF #_w1 THEN "Volume counter"."Control A"."New CV  For ratio check" := 0; END_IF;
   "Volume counter"."Control A"."Current Pulses  For ratio check" := 0 - "Volume counter"."Control A"."New CV  For ratio check";
   "Volume counter"."Volume A"."volume For Ratio check" := "Volume counter"."Control A"."Current Pulses  For ratio check" * "Volume counter"."A".Impulse;
   #_w2 := "AlwaysFALSE" AND "Function Ratio check".Control."metering running" AND "Clock_1Hz" AND NOT "Temp".temp_3[5];   // rising edge of "Clock_1Hz"
   "Temp".temp_3[5] := "Clock_1Hz";
   IF #_w2 THEN
       "Volume counter"."Volume A"."volume For Ratio check" := ("Flowrate".Current."B"/60.0)+"Volume counter"."Volume A"."volume For Ratio check";
   END_IF;
   IF "AlwaysFALSE" AND "Function Ratio check".Control."metering completed" THEN
       "Volume counter"."Volume A"."volume For Ratio check" := 0.0;
   END_IF;
END_REGION

REGION Network 23: B volume During ratio check
   RUNG wire#powerrail
      P_Contact(operand := "Volume counter"."Control B"."Create New CV For ratio check", bit := #temp4)
      Move(in := 0, out1 => "Volume counter"."Control B"."New CV For ratio check")
   END_RUNG
   RUNG wire#powerrail
      Sub(in1 := 0, in2 := "Volume counter"."Control B"."New CV For ratio check", out => "Volume counter"."Control B"."Current Pulses For ratio check")
      Mul(in1 := "Volume counter"."Control B"."Current Pulses For ratio check", in2 := "Volume counter"."B".Impulse, out => "Volume counter"."Volume B"."volume For Ratio check")
   END_RUNG
   RUNG wire#powerrail
      Contact( "AlwaysFALSE" )
      Contact( "Function Ratio check".Control."metering running" )
      P_Contact(operand := "Clock_1Hz", bit := "Temp".temp_3[6])
      { S7_Templates := "SrcType := Real"; S7_Expression := "(IN1/IN2)+IN3" } Calculate(in1 := "Flowrate".Current."B", in2 := 60.0, in3 := "Volume counter"."Volume B"."volume For Ratio check", out => "Volume counter"."Volume B"."volume For Ratio check")
   END_RUNG
   RUNG wire#powerrail
      Contact( "AlwaysFALSE" )
      Contact( "Function Ratio check".Control."metering completed" )
      Move(in := 0.0, out1 => "Volume counter"."Volume B"."volume For Ratio check")
   END_RUNG
   // the same network as SCL:
   #_w1 := "Volume counter"."Control B"."Create New CV For ratio check" AND NOT #temp4;   // rising edge of "Volume counter"."Control B"."Create New CV For ratio check"
   #temp4 := "Volume counter"."Control B"."Create New CV For ratio check";
   IF #_w1 THEN "Volume counter"."Control B"."New CV For ratio check" := 0; END_IF;
   "Volume counter"."Control B"."Current Pulses For ratio check" := 0 - "Volume counter"."Control B"."New CV For ratio check";
   "Volume counter"."Volume B"."volume For Ratio check" := "Volume counter"."Control B"."Current Pulses For ratio check" * "Volume counter"."B".Impulse;
   #_w2 := "AlwaysFALSE" AND "Function Ratio check".Control."metering running" AND "Clock_1Hz" AND NOT "Temp".temp_3[6];   // rising edge of "Clock_1Hz"
   "Temp".temp_3[6] := "Clock_1Hz";
   IF #_w2 THEN
       "Volume counter"."Volume B"."volume For Ratio check" := ("Flowrate".Current."B"/60.0)+"Volume counter"."Volume B"."volume For Ratio check";
   END_IF;
   IF "AlwaysFALSE" AND "Function Ratio check".Control."metering completed" THEN
       "Volume counter"."Volume B"."volume For Ratio check" := 0.0;
   END_IF;
END_REGION
END_ORGANIZATION_BLOCK

FUNCTION "pump RPM" : Void   // FC28, LAD
{ S7_Optimized_Access := 'TRUE' }
VERSION : 0.1
// stored: AutoNumber true, IsIECCheckEnabled false, SetENOAutomatically false, UDAEnableTagReadback false
BEGIN

REGION Network 1 (SCL)
   "RPM".A := ((DINT_TO_REAL("RPM PUMP A")) / "Pump & Flowrate"."Pump A"."speed sensor impulse") * 60.0;
   "RPM".B := ((DINT_TO_REAL("RPM PUMP B")) / "Pump & Flowrate"."Pump B"."speed sensor impulse") * 60.0;

   "RPM"."a selected" := ("RPM"."speed sensor selection A" = 1);
   "RPM"."b selected" := ("RPM"."speed sensor selection B" = 1);
   "RPM"."ab selected" := "RPM"."a selected" OR "RPM"."b selected";
END_REGION
END_FUNCTION

FUNCTION "Re-filling Sequence" : Void   // FC14, LAD
{ S7_Optimized_Access := 'TRUE' }
VERSION : 0.1
// stored: AutoNumber true, IsIECCheckEnabled false, SetENOAutomatically false, UDAEnableTagReadback false
   VAR_TEMP   // added for the SCL form of the ladder/FBD networks
      _w1 : Bool;
      _w2 : Bool;
      _w3 : Bool;
   END_VAR
BEGIN

REGION Network 1
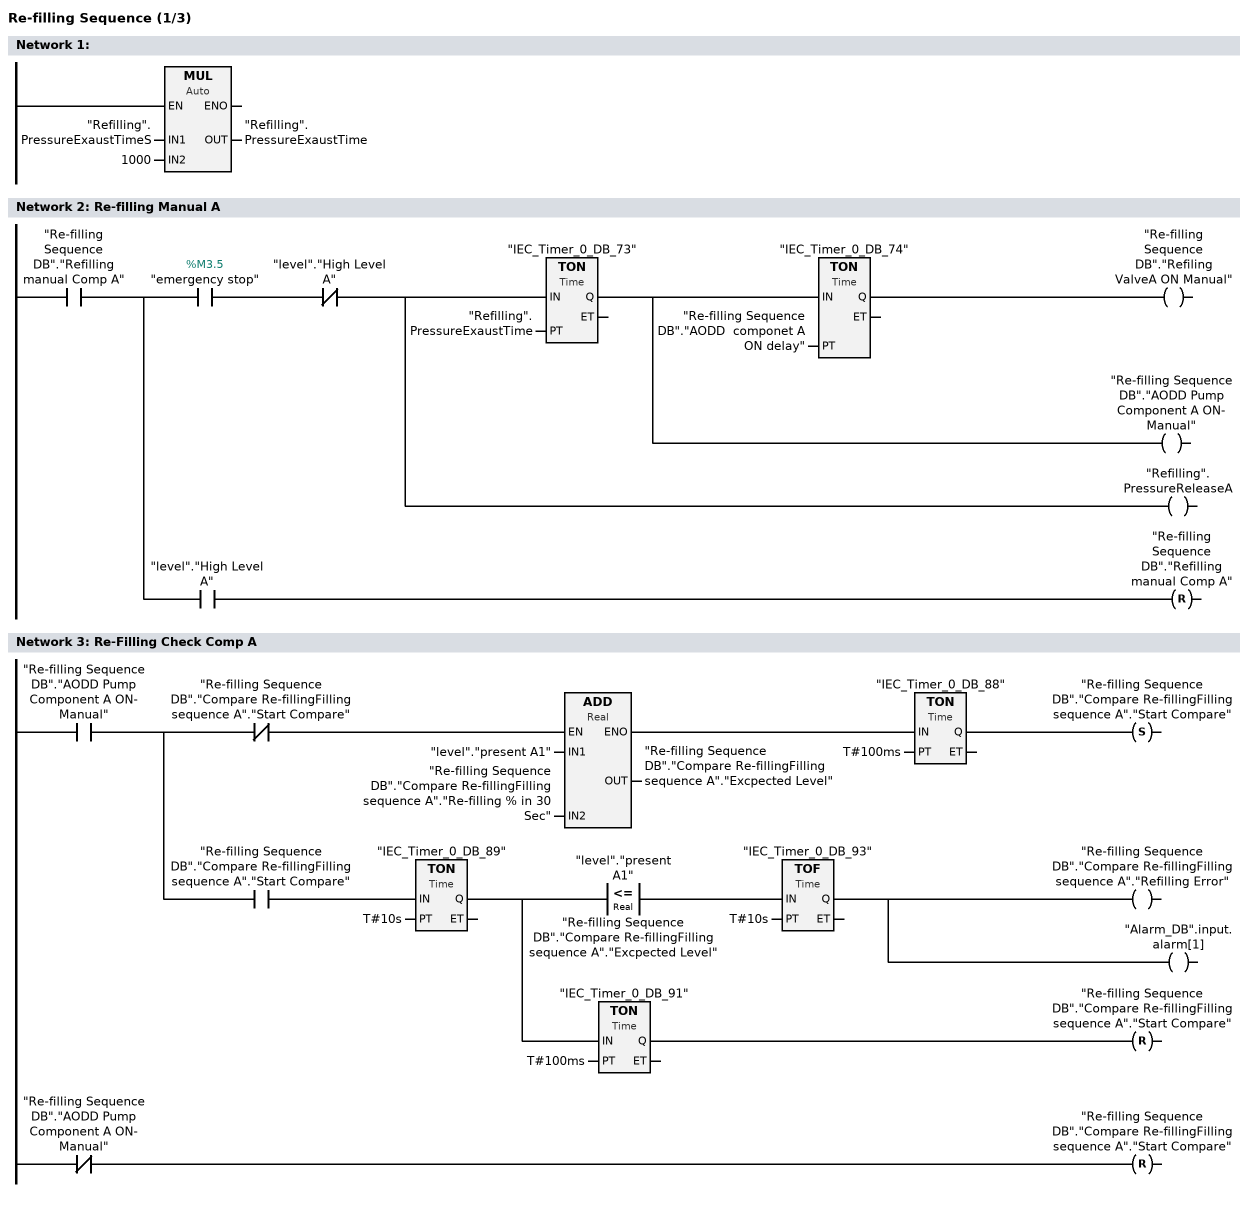
   RUNG wire#powerrail
      Mul(in1 := "Refilling".PressureExaustTimeS, in2 := 1000, out => "Refilling".PressureExaustTime)
   END_RUNG
   // the same network as SCL:
   "Refilling".PressureExaustTime := "Refilling".PressureExaustTimeS * 1000;
END_REGION

REGION Network 2: Re-filling Manual A
   RUNG wire#powerrail
      Contact( "Re-filling Sequence DB"."Refilling manual Comp A" )
      wire#w1
      Contact( "emergency stop" )
      I_Contact( "level"."High Level A" )
      wire#w2
      { S7_Templates := "time_type := Time" } "IEC_Timer_0_DB_73".TON(pt := "Refilling".PressureExaustTime, et =>)
      wire#w3
      { S7_Templates := "time_type := Time" } "IEC_Timer_0_DB_74".TON(pt := "Re-filling Sequence DB"."AODD  componet A  ON delay", et =>)
      Coil( "Re-filling Sequence DB"."Refiling ValveA ON Manual" )
   END_RUNG
   RUNG wire#w3
      Coil( "Re-filling Sequence DB"."AODD Pump Component A ON- Manual" )
   END_RUNG
   RUNG wire#w2
      Coil( "Refilling".PressureReleaseA )
   END_RUNG
   RUNG wire#w1
      Contact( "level"."High Level A" )
      R_Coil( "Re-filling Sequence DB"."Refilling manual Comp A" )
   END_RUNG
   // the same network as SCL:
   #_w1 := "Re-filling Sequence DB"."Refilling manual Comp A" AND "emergency stop" AND NOT "level"."High Level A";
   "IEC_Timer_0_DB_73".TON(IN := #_w1, PT := "Refilling".PressureExaustTime);
   "IEC_Timer_0_DB_74".TON(IN := "IEC_Timer_0_DB_73".Q,
                           PT := "Re-filling Sequence DB"."AODD  componet A  ON delay");
   "Re-filling Sequence DB"."Refiling ValveA ON Manual" := "IEC_Timer_0_DB_74".Q;
   "Re-filling Sequence DB"."AODD Pump Component A ON- Manual" := "IEC_Timer_0_DB_73".Q;
   "Refilling".PressureReleaseA := #_w1;
   IF "Re-filling Sequence DB"."Refilling manual Comp A" AND "level"."High Level A" THEN
       "Re-filling Sequence DB"."Refilling manual Comp A" := FALSE;
   END_IF;
END_REGION

REGION Network 3: Re-Filling Check Comp A
   RUNG wire#powerrail
      Contact( "Re-filling Sequence DB"."AODD Pump Component A ON- Manual" )
      wire#w1
      I_Contact( "Re-filling Sequence DB"."Compare Re-fillingFilling sequence A"."Start Compare" )
      { S7_Templates := "SrcType := Real" } Add(in1 := "level"."present A1", in2 := "Re-filling Sequence DB"."Compare Re-fillingFilling sequence A"."Re-filling % in 30 Sec", out => "Re-filling Sequence DB"."Compare Re-fillingFilling sequence A"."Excpected Level")
      { S7_Templates := "time_type := Time" } "IEC_Timer_0_DB_88".TON(pt := T#100ms, et =>)
      S_Coil( "Re-filling Sequence DB"."Compare Re-fillingFilling sequence A"."Start Compare" )
   END_RUNG
   RUNG wire#w1
      Contact( "Re-filling Sequence DB"."Compare Re-fillingFilling sequence A"."Start Compare" )
      { S7_Templates := "time_type := Time" } "IEC_Timer_0_DB_89".TON(pt := T#10s, et =>)
      wire#w2
      { S7_Templates := "SrcType := Real" } LE_Contact(in1 := "level"."present A1", in2 := "Re-filling Sequence DB"."Compare Re-fillingFilling sequence A"."Excpected Level")
      { S7_Templates := "time_type := Time" } "IEC_Timer_0_DB_93".TOF(pt := T#10s, et =>)
      wire#w3
      Coil( "Re-filling Sequence DB"."Compare Re-fillingFilling sequence A"."Refilling Error" )
   END_RUNG
   RUNG wire#w3
      Coil( "Alarm_DB".input.alarm[1] )
   END_RUNG
   RUNG wire#w2
      { S7_Templates := "time_type := Time" } "IEC_Timer_0_DB_91".TON(pt := T#100ms, et =>)
      R_Coil( "Re-filling Sequence DB"."Compare Re-fillingFilling sequence A"."Start Compare" )
   END_RUNG
   RUNG wire#powerrail
      I_Contact( "Re-filling Sequence DB"."AODD Pump Component A ON- Manual" )
      R_Coil( "Re-filling Sequence DB"."Compare Re-fillingFilling sequence A"."Start Compare" )
   END_RUNG
   // the same network as SCL:
   #_w1 := "Re-filling Sequence DB"."AODD Pump Component A ON- Manual" AND NOT "Re-filling Sequence DB"."Compare Re-fillingFilling sequence A"."Start Compare";
   IF #_w1 THEN
       "Re-filling Sequence DB"."Compare Re-fillingFilling sequence A"."Excpected Level" := "level"."present A1" + "Re-filling Sequence DB"."Compare Re-fillingFilling sequence A"."Re-filling % in 30 Sec";
   END_IF;
   "IEC_Timer_0_DB_88".TON(IN := #_w1, PT := T#100ms);
   IF "IEC_Timer_0_DB_88".Q THEN
       "Re-filling Sequence DB"."Compare Re-fillingFilling sequence A"."Start Compare" := TRUE;
   END_IF;
   "IEC_Timer_0_DB_89".TON(IN := "Re-filling Sequence DB"."AODD Pump Component A ON- Manual" AND "Re-filling Sequence DB"."Compare Re-fillingFilling sequence A"."Start Compare",
                           PT := T#10s);
   "IEC_Timer_0_DB_93".TOF(IN := "IEC_Timer_0_DB_89".Q AND ("level"."present A1" <= "Re-filling Sequence DB"."Compare Re-fillingFilling sequence A"."Excpected Level"),
                           PT := T#10s);
   "Re-filling Sequence DB"."Compare Re-fillingFilling sequence A"."Refilling Error" := "IEC_Timer_0_DB_93".Q;
   "Alarm_DB".input.alarm[1] := "IEC_Timer_0_DB_93".Q;
   "IEC_Timer_0_DB_91".TON(IN := "IEC_Timer_0_DB_89".Q, PT := T#100ms);
   IF "IEC_Timer_0_DB_91".Q THEN
       "Re-filling Sequence DB"."Compare Re-fillingFilling sequence A"."Start Compare" := FALSE;
   END_IF;
   IF NOT "Re-filling Sequence DB"."AODD Pump Component A ON- Manual" THEN
       "Re-filling Sequence DB"."Compare Re-fillingFilling sequence A"."Start Compare" := FALSE;
   END_IF;
END_REGION

REGION Network 4: Re-filling Manual B
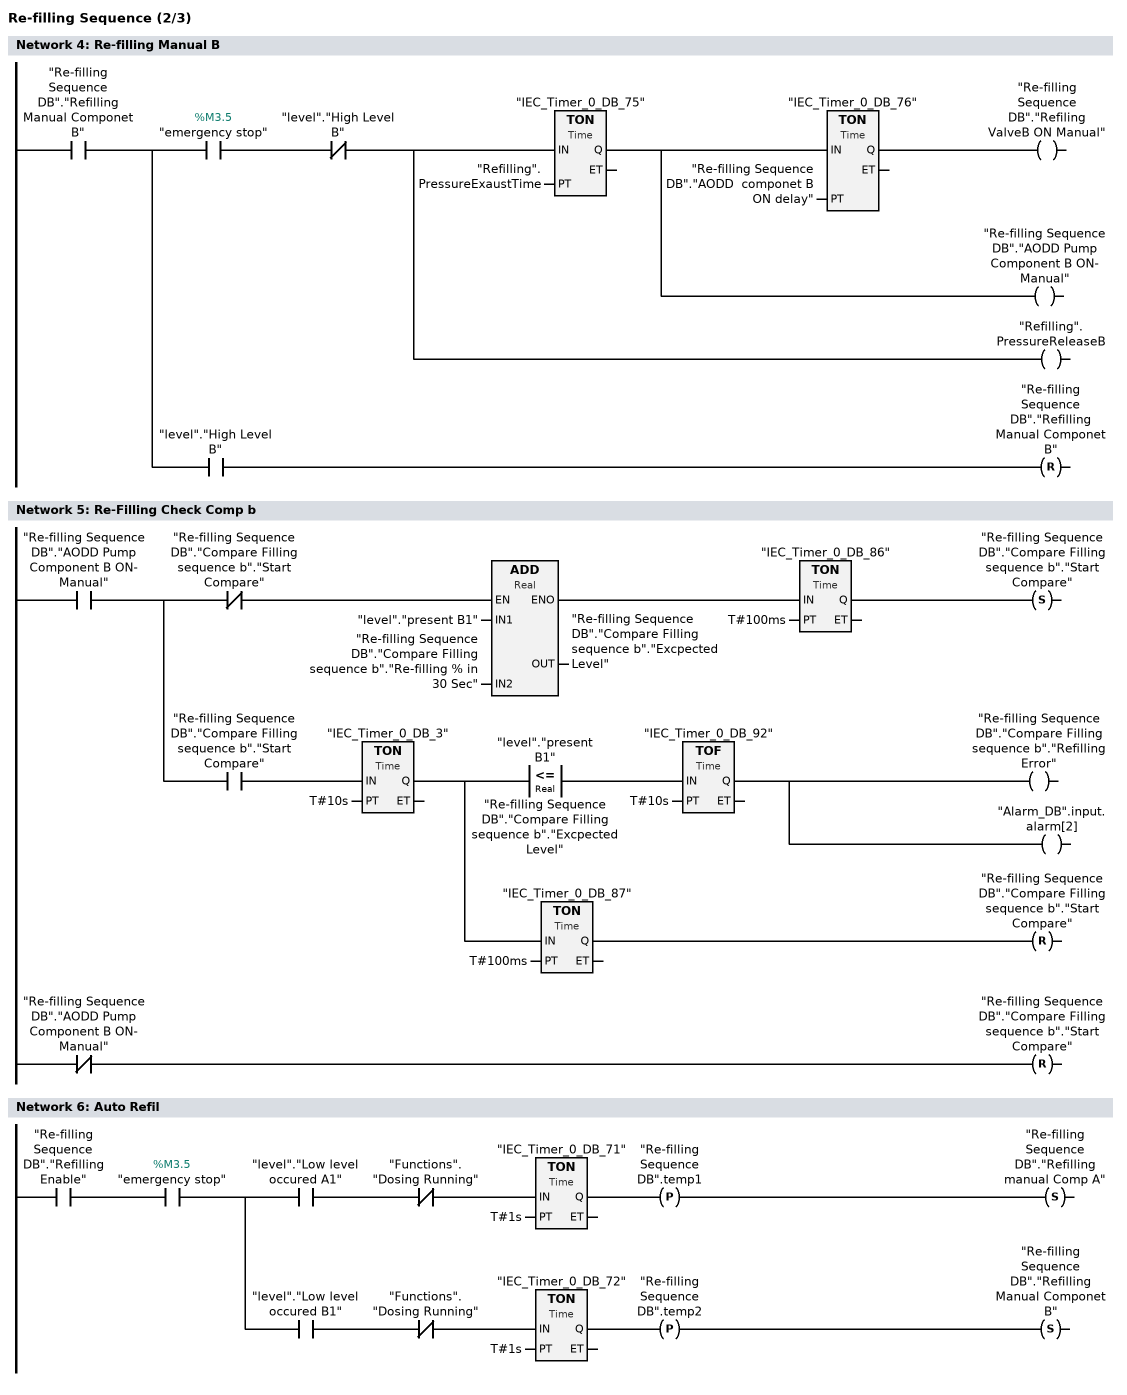
   RUNG wire#powerrail
      Contact( "Re-filling Sequence DB"."Refilling Manual Componet B" )
      wire#w1
      Contact( "emergency stop" )
      I_Contact( "level"."High Level B" )
      wire#w2
      { S7_Templates := "time_type := Time" } "IEC_Timer_0_DB_75".TON(pt := "Refilling".PressureExaustTime, et =>)
      wire#w3
      { S7_Templates := "time_type := Time" } "IEC_Timer_0_DB_76".TON(pt := "Re-filling Sequence DB"."AODD  componet B  ON delay", et =>)
      Coil( "Re-filling Sequence DB"."Refiling ValveB ON Manual" )
   END_RUNG
   RUNG wire#w3
      Coil( "Re-filling Sequence DB"."AODD Pump Component B ON- Manual" )
   END_RUNG
   RUNG wire#w2
      Coil( "Refilling".PressureReleaseB )
   END_RUNG
   RUNG wire#w1
      Contact( "level"."High Level B" )
      R_Coil( "Re-filling Sequence DB"."Refilling Manual Componet B" )
   END_RUNG
   // the same network as SCL:
   #_w1 := "Re-filling Sequence DB"."Refilling Manual Componet B" AND "emergency stop" AND NOT "level"."High Level B";
   "IEC_Timer_0_DB_75".TON(IN := #_w1, PT := "Refilling".PressureExaustTime);
   "IEC_Timer_0_DB_76".TON(IN := "IEC_Timer_0_DB_75".Q,
                           PT := "Re-filling Sequence DB"."AODD  componet B  ON delay");
   "Re-filling Sequence DB"."Refiling ValveB ON Manual" := "IEC_Timer_0_DB_76".Q;
   "Re-filling Sequence DB"."AODD Pump Component B ON- Manual" := "IEC_Timer_0_DB_75".Q;
   "Refilling".PressureReleaseB := #_w1;
   IF "Re-filling Sequence DB"."Refilling Manual Componet B" AND "level"."High Level B" THEN
       "Re-filling Sequence DB"."Refilling Manual Componet B" := FALSE;
   END_IF;
END_REGION

REGION Network 5: Re-Filling Check Comp b
   RUNG wire#powerrail
      Contact( "Re-filling Sequence DB"."AODD Pump Component B ON- Manual" )
      wire#w1
      I_Contact( "Re-filling Sequence DB"."Compare Filling sequence b"."Start Compare" )
      { S7_Templates := "SrcType := Real" } Add(in1 := "level"."present B1", in2 := "Re-filling Sequence DB"."Compare Filling sequence b"."Re-filling % in 30 Sec", out => "Re-filling Sequence DB"."Compare Filling sequence b"."Excpected Level")
      { S7_Templates := "time_type := Time" } "IEC_Timer_0_DB_86".TON(pt := T#100ms, et =>)
      S_Coil( "Re-filling Sequence DB"."Compare Filling sequence b"."Start Compare" )
   END_RUNG
   RUNG wire#w1
      Contact( "Re-filling Sequence DB"."Compare Filling sequence b"."Start Compare" )
      { S7_Templates := "time_type := Time" } "IEC_Timer_0_DB_3".TON(pt := T#10s, et =>)
      wire#w2
      { S7_Templates := "SrcType := Real" } LE_Contact(in1 := "level"."present B1", in2 := "Re-filling Sequence DB"."Compare Filling sequence b"."Excpected Level")
      { S7_Templates := "time_type := Time" } "IEC_Timer_0_DB_92".TOF(pt := T#10s, et =>)
      wire#w3
      Coil( "Re-filling Sequence DB"."Compare Filling sequence b"."Refilling Error" )
   END_RUNG
   RUNG wire#w3
      Coil( "Alarm_DB".input.alarm[2] )
   END_RUNG
   RUNG wire#w2
      { S7_Templates := "time_type := Time" } "IEC_Timer_0_DB_87".TON(pt := T#100ms, et =>)
      R_Coil( "Re-filling Sequence DB"."Compare Filling sequence b"."Start Compare" )
   END_RUNG
   RUNG wire#powerrail
      I_Contact( "Re-filling Sequence DB"."AODD Pump Component B ON- Manual" )
      R_Coil( "Re-filling Sequence DB"."Compare Filling sequence b"."Start Compare" )
   END_RUNG
   // the same network as SCL:
   #_w1 := "Re-filling Sequence DB"."AODD Pump Component B ON- Manual" AND NOT "Re-filling Sequence DB"."Compare Filling sequence b"."Start Compare";
   IF #_w1 THEN
       "Re-filling Sequence DB"."Compare Filling sequence b"."Excpected Level" := "level"."present B1" + "Re-filling Sequence DB"."Compare Filling sequence b"."Re-filling % in 30 Sec";
   END_IF;
   "IEC_Timer_0_DB_86".TON(IN := #_w1, PT := T#100ms);
   IF "IEC_Timer_0_DB_86".Q THEN
       "Re-filling Sequence DB"."Compare Filling sequence b"."Start Compare" := TRUE;
   END_IF;
   "IEC_Timer_0_DB_3".TON(IN := "Re-filling Sequence DB"."AODD Pump Component B ON- Manual" AND "Re-filling Sequence DB"."Compare Filling sequence b"."Start Compare",
                          PT := T#10s);
   "IEC_Timer_0_DB_92".TOF(IN := "IEC_Timer_0_DB_3".Q AND ("level"."present B1" <= "Re-filling Sequence DB"."Compare Filling sequence b"."Excpected Level"),
                           PT := T#10s);
   "Re-filling Sequence DB"."Compare Filling sequence b"."Refilling Error" := "IEC_Timer_0_DB_92".Q;
   "Alarm_DB".input.alarm[2] := "IEC_Timer_0_DB_92".Q;
   "IEC_Timer_0_DB_87".TON(IN := "IEC_Timer_0_DB_3".Q, PT := T#100ms);
   IF "IEC_Timer_0_DB_87".Q THEN
       "Re-filling Sequence DB"."Compare Filling sequence b"."Start Compare" := FALSE;
   END_IF;
   IF NOT "Re-filling Sequence DB"."AODD Pump Component B ON- Manual" THEN
       "Re-filling Sequence DB"."Compare Filling sequence b"."Start Compare" := FALSE;
   END_IF;
END_REGION

REGION Network 6: Auto Refil
   RUNG wire#powerrail
      Contact( "Re-filling Sequence DB"."Refilling Enable" )
      Contact( "emergency stop" )
      wire#w1
      Contact( "level"."Low level occured A1" )
      I_Contact( "Functions"."Dosing Running" )
      { S7_Templates := "time_type := Time" } "IEC_Timer_0_DB_71".TON(pt := T#1s, et =>)
      P_Trig( "Re-filling Sequence DB".temp1 )
      S_Coil( "Re-filling Sequence DB"."Refilling manual Comp A" )
   END_RUNG
   RUNG wire#w1
      Contact( "level"."Low level occured B1" )
      I_Contact( "Functions"."Dosing Running" )
      { S7_Templates := "time_type := Time" } "IEC_Timer_0_DB_72".TON(pt := T#1s, et =>)
      P_Trig( "Re-filling Sequence DB".temp2 )
      S_Coil( "Re-filling Sequence DB"."Refilling Manual Componet B" )
   END_RUNG
   // the same network as SCL:
   #_w1 := "Re-filling Sequence DB"."Refilling Enable" AND "emergency stop";
   "IEC_Timer_0_DB_71".TON(IN := #_w1 AND "level"."Low level occured A1" AND NOT "Functions"."Dosing Running",
                           PT := T#1s);
   #_w2 := "IEC_Timer_0_DB_71".Q AND NOT "Re-filling Sequence DB".temp1;   // rising edge
   "Re-filling Sequence DB".temp1 := "IEC_Timer_0_DB_71".Q;
   IF #_w2 THEN "Re-filling Sequence DB"."Refilling manual Comp A" := TRUE; END_IF;
   "IEC_Timer_0_DB_72".TON(IN := #_w1 AND "level"."Low level occured B1" AND NOT "Functions"."Dosing Running",
                           PT := T#1s);
   #_w3 := "IEC_Timer_0_DB_72".Q AND NOT "Re-filling Sequence DB".temp2;   // rising edge
   "Re-filling Sequence DB".temp2 := "IEC_Timer_0_DB_72".Q;
   IF #_w3 THEN "Re-filling Sequence DB"."Refilling Manual Componet B" := TRUE; END_IF;
END_REGION

REGION Network 7: Auto reffil reset
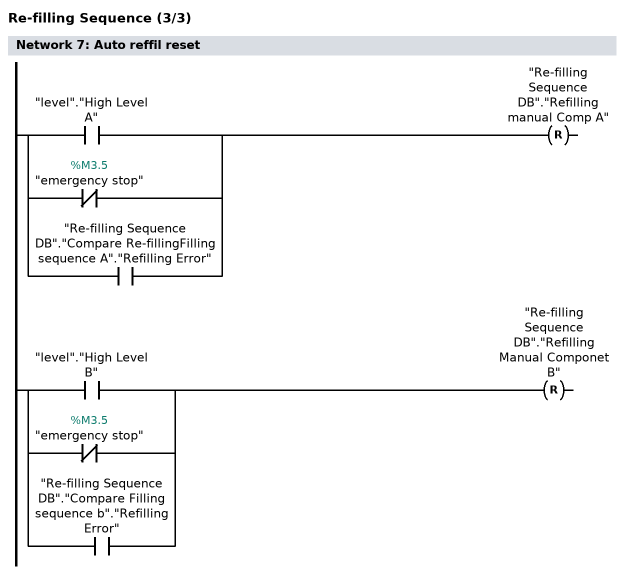
   RUNG wire#powerrail
      Contact( "level"."High Level A" )
      wire#w1
      R_Coil( "Re-filling Sequence DB"."Refilling manual Comp A" )
   END_RUNG
   RUNG wire#powerrail
      I_Contact( "emergency stop" )
   END_RUNG wire#w1
   RUNG wire#powerrail
      Contact( "Re-filling Sequence DB"."Compare Re-fillingFilling sequence A"."Refilling Error" )
   END_RUNG wire#w1
   RUNG wire#powerrail
      Contact( "level"."High Level B" )
      wire#w2
      R_Coil( "Re-filling Sequence DB"."Refilling Manual Componet B" )
   END_RUNG
   RUNG wire#powerrail
      I_Contact( "emergency stop" )
   END_RUNG wire#w2
   RUNG wire#powerrail
      Contact( "Re-filling Sequence DB"."Compare Filling sequence b"."Refilling Error" )
   END_RUNG wire#w2
   // the same network as SCL:
   IF "level"."High Level A" OR NOT "emergency stop" OR "Re-filling Sequence DB"."Compare Re-fillingFilling sequence A"."Refilling Error" THEN
       "Re-filling Sequence DB"."Refilling manual Comp A" := FALSE;
   END_IF;
   IF "level"."High Level B" OR NOT "emergency stop" OR "Re-filling Sequence DB"."Compare Filling sequence b"."Refilling Error" THEN
       "Re-filling Sequence DB"."Refilling Manual Componet B" := FALSE;
   END_IF;
END_REGION
END_FUNCTION

FUNCTION "Pump Management" : Void   // FC44, LAD
{ S7_Optimized_Access := 'TRUE' }
VERSION : 0.1
// stored: AutoNumber false, IsIECCheckEnabled false, SetENOAutomatically false, UDAEnableTagReadback false
   VAR_TEMP
      mbit1 : Bool;
   END_VAR
BEGIN

REGION Network 1
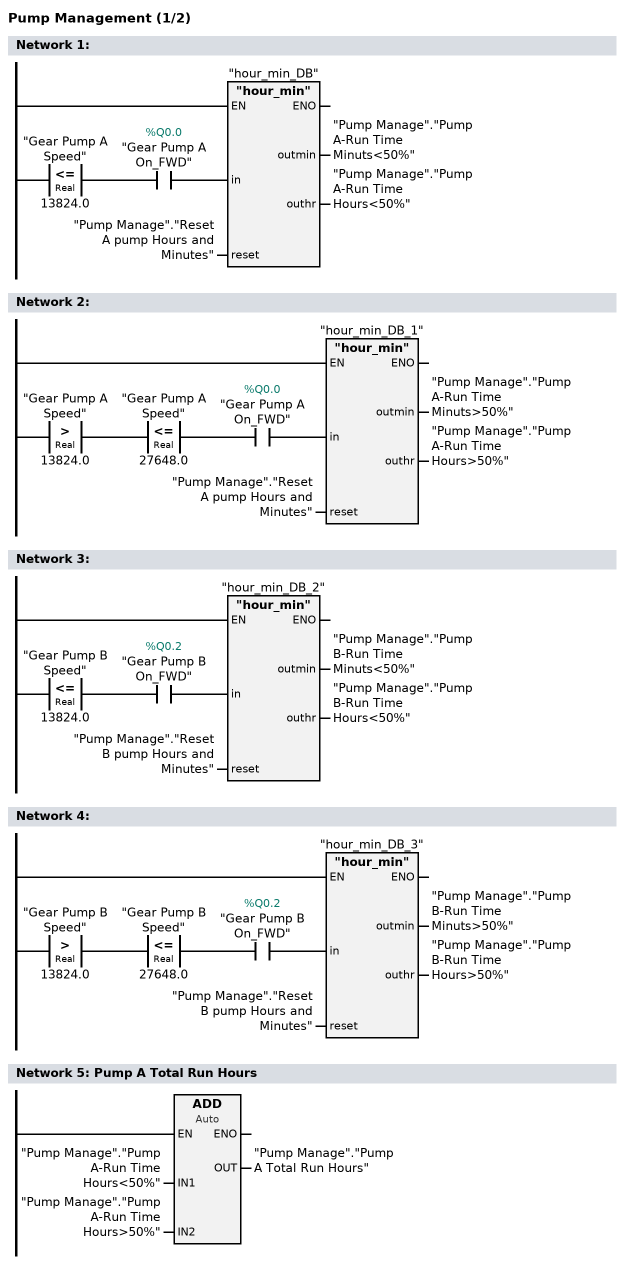
   RUNG wire#powerrail
      "hour_min_DB"(in := wire#w1, reset := "Pump Manage"."Reset A pump Hours and Minutes", outmin => "Pump Manage"."Pump A-Run Time Minuts<50%", outhr => "Pump Manage"."Pump A-Run Time Hours<50%")
   END_RUNG
   RUNG wire#powerrail
      { S7_Templates := "SrcType := Real" } LE_Contact(in1 := "Gear Pump A Speed", in2 := 13824.0)
      Contact( "Gear Pump A On_FWD" )
   END_RUNG wire#w1
   // the same network as SCL:
   "hour_min_DB"(in := ("Gear Pump A Speed" <= 13824.0) AND "Gear Pump A On_FWD",   // "hour_min"
                 reset := "Pump Manage"."Reset A pump Hours and Minutes",
                 outmin => "Pump Manage"."Pump A-Run Time Minuts<50%",
                 outhr => "Pump Manage"."Pump A-Run Time Hours<50%");
END_REGION

REGION Network 2
   RUNG wire#powerrail
      "hour_min_DB_1"(in := wire#w1, reset := "Pump Manage"."Reset A pump Hours and Minutes", outmin => "Pump Manage"."Pump A-Run Time Minuts>50%", outhr => "Pump Manage"."Pump A-Run Time Hours>50%")
   END_RUNG
   RUNG wire#powerrail
      { S7_Templates := "SrcType := Real" } GT_Contact(in1 := "Gear Pump A Speed", in2 := 13824.0)
      { S7_Templates := "SrcType := Real" } LE_Contact(in1 := "Gear Pump A Speed", in2 := 27648.0)
      Contact( "Gear Pump A On_FWD" )
   END_RUNG wire#w1
   // the same network as SCL:
   "hour_min_DB_1"(in := ("Gear Pump A Speed" > 13824.0) AND ("Gear Pump A Speed" <= 27648.0) AND "Gear Pump A On_FWD",   // "hour_min"
                   reset := "Pump Manage"."Reset A pump Hours and Minutes",
                   outmin => "Pump Manage"."Pump A-Run Time Minuts>50%",
                   outhr => "Pump Manage"."Pump A-Run Time Hours>50%");
END_REGION

REGION Network 3
   RUNG wire#powerrail
      "hour_min_DB_2"(in := wire#w1, reset := "Pump Manage"."Reset B pump Hours and Minutes", outmin => "Pump Manage"."Pump B-Run Time Minuts<50%", outhr => "Pump Manage"."Pump B-Run Time Hours<50%")
   END_RUNG
   RUNG wire#powerrail
      { S7_Templates := "SrcType := Real" } LE_Contact(in1 := "Gear Pump B Speed", in2 := 13824.0)
      Contact( "Gear Pump B On_FWD" )
   END_RUNG wire#w1
   // the same network as SCL:
   "hour_min_DB_2"(in := ("Gear Pump B Speed" <= 13824.0) AND "Gear Pump B On_FWD",   // "hour_min"
                   reset := "Pump Manage"."Reset B pump Hours and Minutes",
                   outmin => "Pump Manage"."Pump B-Run Time Minuts<50%",
                   outhr => "Pump Manage"."Pump B-Run Time Hours<50%");
END_REGION

REGION Network 4
   RUNG wire#powerrail
      "hour_min_DB_3"(in := wire#w1, reset := "Pump Manage"."Reset B pump Hours and Minutes", outmin => "Pump Manage"."Pump B-Run Time Minuts>50%", outhr => "Pump Manage"."Pump B-Run Time Hours>50%")
   END_RUNG
   RUNG wire#powerrail
      { S7_Templates := "SrcType := Real" } GT_Contact(in1 := "Gear Pump B Speed", in2 := 13824.0)
      { S7_Templates := "SrcType := Real" } LE_Contact(in1 := "Gear Pump B Speed", in2 := 27648.0)
      Contact( "Gear Pump B On_FWD" )
   END_RUNG wire#w1
   // the same network as SCL:
   "hour_min_DB_3"(in := ("Gear Pump B Speed" > 13824.0) AND ("Gear Pump B Speed" <= 27648.0) AND "Gear Pump B On_FWD",   // "hour_min"
                   reset := "Pump Manage"."Reset B pump Hours and Minutes",
                   outmin => "Pump Manage"."Pump B-Run Time Minuts>50%",
                   outhr => "Pump Manage"."Pump B-Run Time Hours>50%");
END_REGION

REGION Network 5: Pump A Total Run Hours
   RUNG wire#powerrail
      Add(in1 := "Pump Manage"."Pump A-Run Time Hours<50%", in2 := "Pump Manage"."Pump A-Run Time Hours>50%", out => "Pump Manage"."Pump A Total Run Hours")
   END_RUNG
   // the same network as SCL:
   "Pump Manage"."Pump A Total Run Hours" := "Pump Manage"."Pump A-Run Time Hours<50%" + "Pump Manage"."Pump A-Run Time Hours>50%";
END_REGION

REGION Network 6: Pump A Total Run Minutes
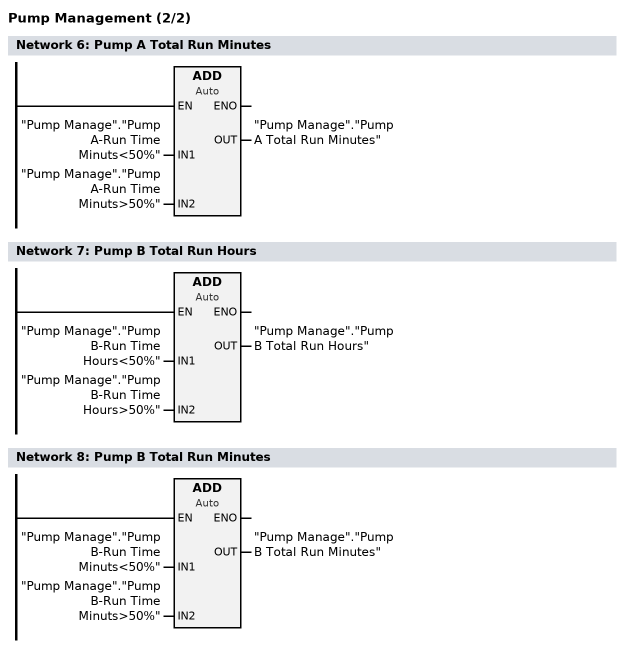
   RUNG wire#powerrail
      Add(in1 := "Pump Manage"."Pump A-Run Time Minuts<50%", in2 := "Pump Manage"."Pump A-Run Time Minuts>50%", out => "Pump Manage"."Pump A Total Run Minutes")
   END_RUNG
   // the same network as SCL:
   "Pump Manage"."Pump A Total Run Minutes" := "Pump Manage"."Pump A-Run Time Minuts<50%" + "Pump Manage"."Pump A-Run Time Minuts>50%";
END_REGION

REGION Network 7: Pump B Total Run Hours
   RUNG wire#powerrail
      Add(in1 := "Pump Manage"."Pump B-Run Time Hours<50%", in2 := "Pump Manage"."Pump B-Run Time Hours>50%", out => "Pump Manage"."Pump B Total Run Hours")
   END_RUNG
   // the same network as SCL:
   "Pump Manage"."Pump B Total Run Hours" := "Pump Manage"."Pump B-Run Time Hours<50%" + "Pump Manage"."Pump B-Run Time Hours>50%";
END_REGION

REGION Network 8: Pump B Total Run Minutes
   RUNG wire#powerrail
      Add(in1 := "Pump Manage"."Pump B-Run Time Minuts<50%", in2 := "Pump Manage"."Pump B-Run Time Minuts>50%", out => "Pump Manage"."Pump B Total Run Minutes")
   END_RUNG
   // the same network as SCL:
   "Pump Manage"."Pump B Total Run Minutes" := "Pump Manage"."Pump B-Run Time Minuts<50%" + "Pump Manage"."Pump B-Run Time Minuts>50%";
END_REGION
END_FUNCTION

FUNCTION_BLOCK "hour_min"   // FB6, LAD
{ S7_Optimized_Access := 'TRUE' }
VERSION : 0.1
// stored: AutoNumber true, IsIECCheckEnabled false, IsRetainMemResEnabled false, MemoryReserve 100, SetENOAutomatically false, UDAEnableTagReadback false
   VAR_INPUT
      in : Bool;
      reset : Bool;
   END_VAR
   VAR_OUTPUT
      outmin : Int;
      outhr : Int;
   END_VAR
   VAR RETAIN
      insec : Int;
   END_VAR
   VAR
      temp : Bool;
   END_VAR
   VAR_TEMP   // added for the SCL form of the ladder/FBD networks
      _w1 : Bool;
   END_VAR
BEGIN

REGION Network 1
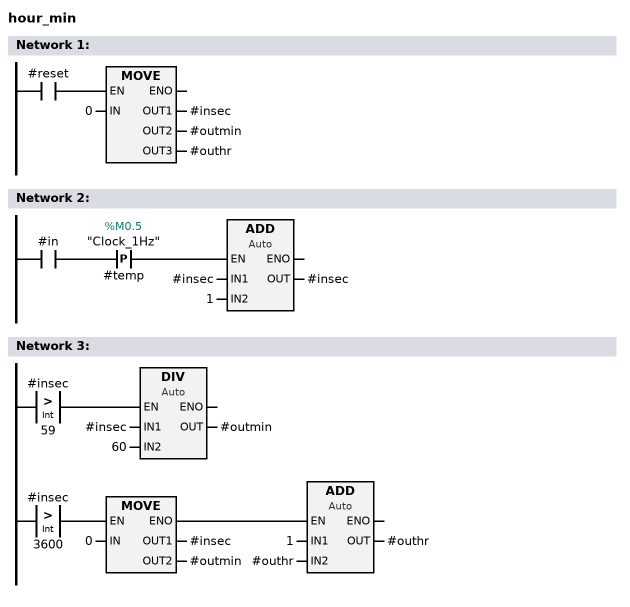
   RUNG wire#powerrail
      Contact( #reset )
      Move(in := 0, out1 => #insec, out2 => #outmin, out3 => #outhr)
   END_RUNG
   // the same network as SCL:
   IF #reset THEN
       #insec := 0;
       #outmin := 0;
       #outhr := 0;
   END_IF;
END_REGION

REGION Network 2
   RUNG wire#powerrail
      Contact( #in )
      P_Contact(operand := "Clock_1Hz", bit := #temp)
      Add(in1 := #insec, in2 := 1, out => #insec)
   END_RUNG
   // the same network as SCL:
   #_w1 := #in AND "Clock_1Hz" AND NOT #temp;   // rising edge of "Clock_1Hz"
   #temp := "Clock_1Hz";
   IF #_w1 THEN #insec := #insec + 1; END_IF;
END_REGION

REGION Network 3
   RUNG wire#powerrail
      { S7_Templates := "SrcType := Int" } GT_Contact(in1 := #insec, in2 := 59)
      Div(in1 := #insec, in2 := 60, out => #outmin)
   END_RUNG
   RUNG wire#powerrail
      { S7_Templates := "SrcType := Int" } GT_Contact(in1 := #insec, in2 := 3600)
      Move(in := 0, out1 => #insec, out2 => #outmin)
      Add(in1 := 1, in2 := #outhr, out => #outhr)
   END_RUNG
   // the same network as SCL:
   IF #insec > 59 THEN #outmin := #insec / 60; END_IF;
   #_w1 := #insec > 3600;
   IF #_w1 THEN
       #insec := 0;
       #outmin := 0;
       #outhr := 1 + #outhr;
   END_IF;
END_REGION
END_FUNCTION_BLOCK

FUNCTION "potlife&regenaration" : Void   // FC22, LAD
{ S7_Optimized_Access := 'TRUE' }
VERSION : 0.1
// stored: AutoNumber true, IsIECCheckEnabled false, SetENOAutomatically false, UDAEnableTagReadback false
   VAR_TEMP
      temp2 : Bool;
   END_VAR
   VAR_TEMP   // added for the SCL form of the ladder/FBD networks
      _w1 : Bool;
   END_VAR
BEGIN

REGION Network 1: regeneration selection
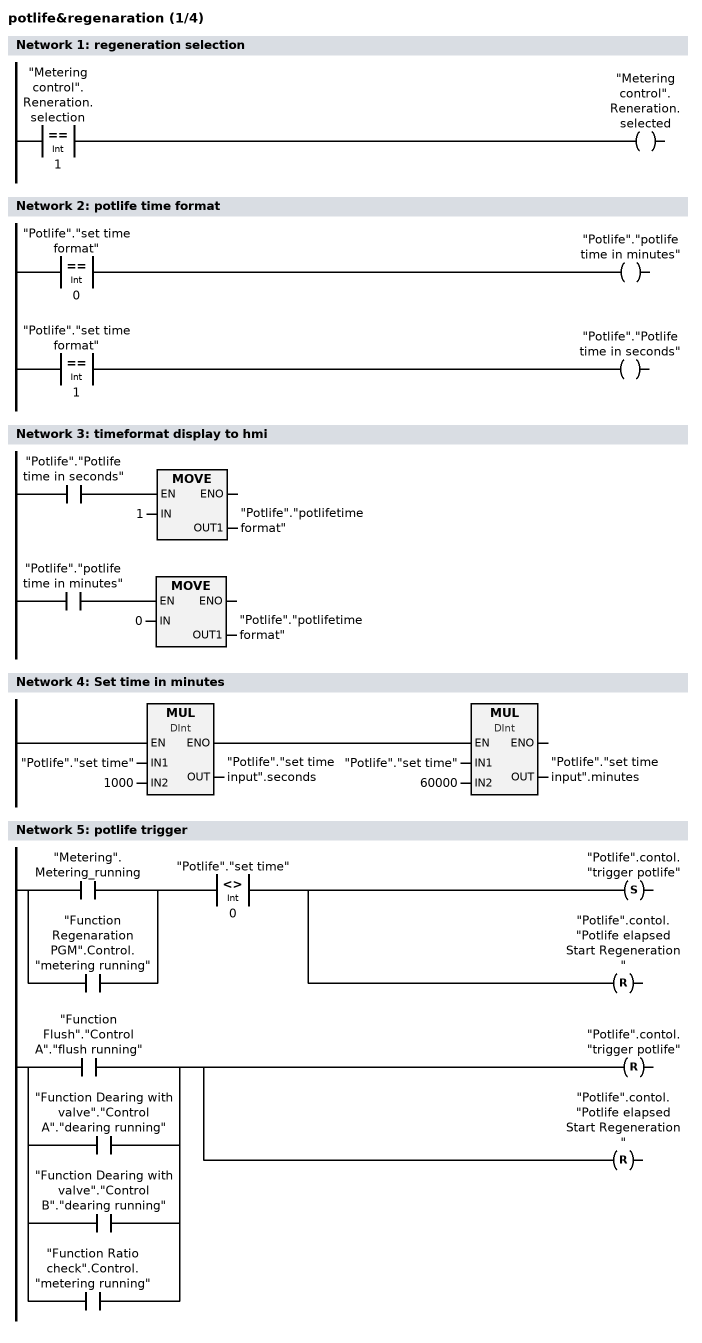
   RUNG wire#powerrail
      { S7_Templates := "SrcType := Int" } EQ_Contact(in1 := "Metering control".Reneration.selection, in2 := 1)
      Coil( "Metering control".Reneration.selected )
   END_RUNG
   // the same network as SCL:
   "Metering control".Reneration.selected := "Metering control".Reneration.selection = 1;
END_REGION

REGION Network 2: potlife time format
   RUNG wire#powerrail
      { S7_Templates := "SrcType := Int" } EQ_Contact(in1 := "Potlife"."set time format", in2 := 0)
      Coil( "Potlife"."potlife time in minutes" )
   END_RUNG
   RUNG wire#powerrail
      { S7_Templates := "SrcType := Int" } EQ_Contact(in1 := "Potlife"."set time format", in2 := 1)
      Coil( "Potlife"."Potlife time in seconds" )
   END_RUNG
   // the same network as SCL:
   "Potlife"."potlife time in minutes" := "Potlife"."set time format" = 0;
   "Potlife"."Potlife time in seconds" := "Potlife"."set time format" = 1;
END_REGION

REGION Network 3: timeformat display to hmi
   RUNG wire#powerrail
      Contact( "Potlife"."Potlife time in seconds" )
      Move(in := 1, out1 => "Potlife"."potlifetime format")
   END_RUNG
   RUNG wire#powerrail
      Contact( "Potlife"."potlife time in minutes" )
      Move(in := 0, out1 => "Potlife"."potlifetime format")
   END_RUNG
   // the same network as SCL:
   IF "Potlife"."Potlife time in seconds" THEN "Potlife"."potlifetime format" := 1; END_IF;
   IF "Potlife"."potlife time in minutes" THEN "Potlife"."potlifetime format" := 0; END_IF;
END_REGION

REGION Network 4: Set time in minutes
   RUNG wire#powerrail
      { S7_Templates := "SrcType := DInt" } Mul(in1 := "Potlife"."set time", in2 := 1000, out => "Potlife"."set time input".seconds)
      { S7_Templates := "SrcType := DInt" } Mul(in1 := "Potlife"."set time", in2 := 60000, out => "Potlife"."set time input".minutes)
   END_RUNG
   // the same network as SCL:
   "Potlife"."set time input".seconds := "Potlife"."set time" * 1000;
   "Potlife"."set time input".minutes := "Potlife"."set time" * 60000;
END_REGION

REGION Network 5: potlife trigger
   RUNG wire#powerrail
      Contact( "Metering".Metering_running )
      wire#w1
      { S7_Templates := "SrcType := Int" } NE_Contact(in1 := "Potlife"."set time", in2 := 0)
      wire#w2
      S_Coil( "Potlife".contol."trigger potlife" )
   END_RUNG
   RUNG wire#powerrail
      Contact( "Function Regenaration PGM".Control."metering running" )
   END_RUNG wire#w1
   RUNG wire#w2
      R_Coil( "Potlife".contol."Potlife elapsed Start Regeneration" )
   END_RUNG
   RUNG wire#powerrail
      Contact( "Function Flush"."Control A"."flush running" )
      wire#w3
      R_Coil( "Potlife".contol."trigger potlife" )
   END_RUNG
   RUNG wire#powerrail
      Contact( "Function Dearing with valve"."Control A"."dearing running" )
   END_RUNG wire#w3
   RUNG wire#powerrail
      Contact( "Function Dearing with valve"."Control B"."dearing running" )
   END_RUNG wire#w3
   RUNG wire#powerrail
      Contact( "Function Ratio check".Control."metering running" )
   END_RUNG wire#w3
   RUNG wire#w3
      R_Coil( "Potlife".contol."Potlife elapsed Start Regeneration" )
   END_RUNG
   // the same network as SCL:
   IF ("Metering".Metering_running OR "Function Regenaration PGM".Control."metering running") AND ("Potlife"."set time" <> 0) THEN
       "Potlife".contol."trigger potlife" := TRUE;
       "Potlife".contol."Potlife elapsed Start Regeneration" := FALSE;
   END_IF;
   IF "Function Flush"."Control A"."flush running" OR "Function Dearing with valve"."Control A"."dearing running" OR "Function Dearing with valve"."Control B"."dearing running" OR "Function Ratio check".Control."metering running" THEN
       "Potlife".contol."trigger potlife" := FALSE;
       "Potlife".contol."Potlife elapsed Start Regeneration" := FALSE;
   END_IF;
END_REGION

REGION Network 6
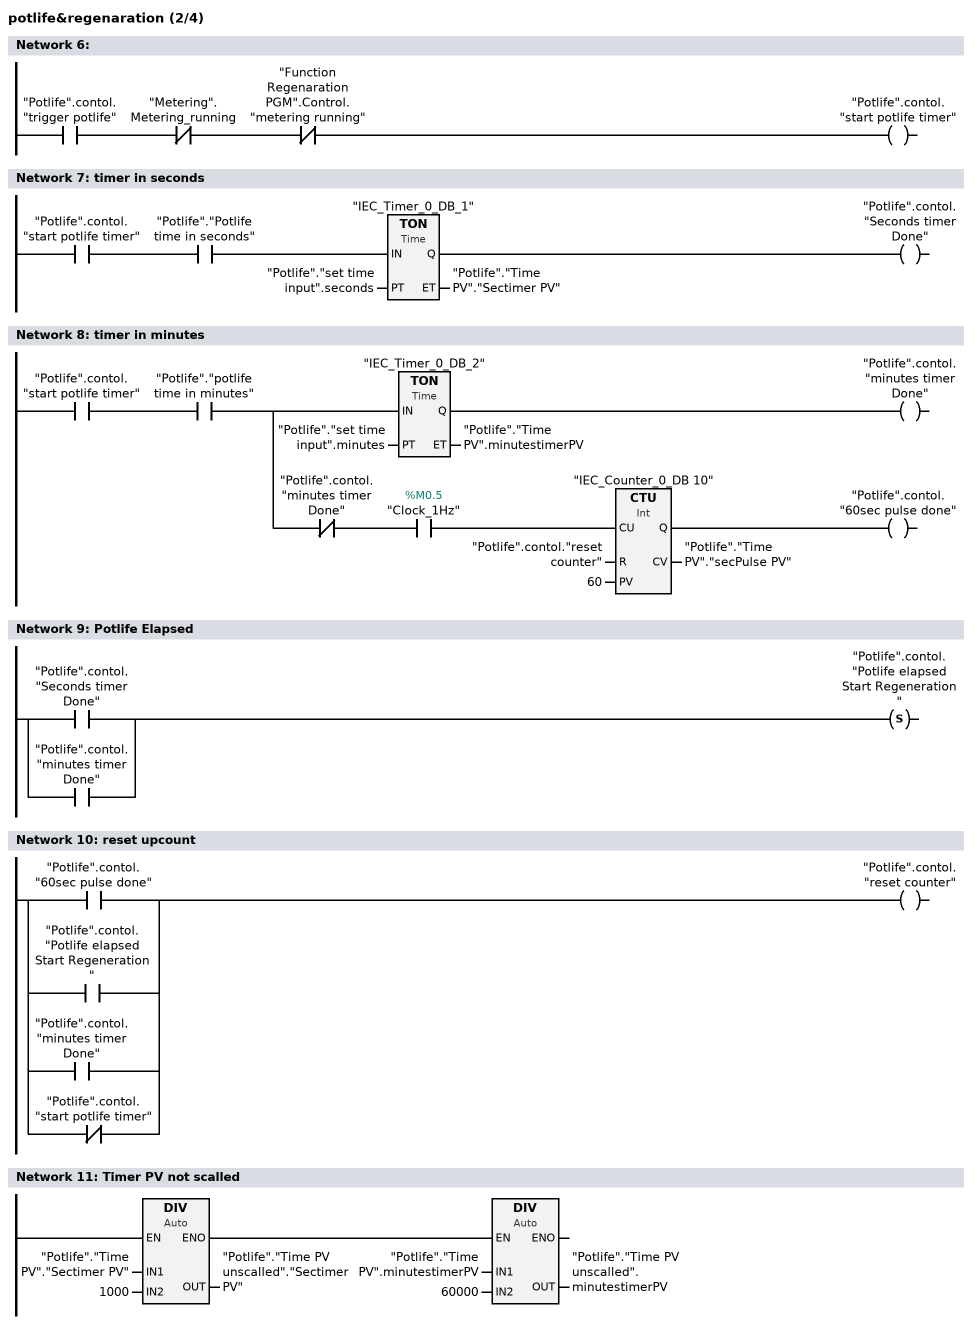
   RUNG wire#powerrail
      Contact( "Potlife".contol."trigger potlife" )
      I_Contact( "Metering".Metering_running )
      I_Contact( "Function Regenaration PGM".Control."metering running" )
      Coil( "Potlife".contol."start potlife timer" )
   END_RUNG
   // the same network as SCL:
   "Potlife".contol."start potlife timer" := "Potlife".contol."trigger potlife" AND NOT "Metering".Metering_running AND NOT "Function Regenaration PGM".Control."metering running";
END_REGION

REGION Network 7: timer in seconds
   RUNG wire#powerrail
      Contact( "Potlife".contol."start potlife timer" )
      Contact( "Potlife"."Potlife time in seconds" )
      { S7_Templates := "time_type := Time" } "IEC_Timer_0_DB_1".TON(pt := "Potlife"."set time input".seconds, et => "Potlife"."Time PV"."Sectimer PV")
      Coil( "Potlife".contol."Seconds timer Done" )
   END_RUNG
   // the same network as SCL:
   "IEC_Timer_0_DB_1".TON(IN := "Potlife".contol."start potlife timer" AND "Potlife"."Potlife time in seconds",
                          PT := "Potlife"."set time input".seconds,
                          ET => "Potlife"."Time PV"."Sectimer PV");
   "Potlife".contol."Seconds timer Done" := "IEC_Timer_0_DB_1".Q;
END_REGION

REGION Network 8: timer in minutes
   RUNG wire#powerrail
      Contact( "Potlife".contol."start potlife timer" )
      Contact( "Potlife"."potlife time in minutes" )
      wire#w1
      { S7_Templates := "time_type := Time" } "IEC_Timer_0_DB_2".TON(pt := "Potlife"."set time input".minutes, et => "Potlife"."Time PV".minutestimerPV)
      Coil( "Potlife".contol."minutes timer Done" )
   END_RUNG
   RUNG wire#w1
      I_Contact( "Potlife".contol."minutes timer Done" )
      Contact( "Clock_1Hz" )
      { S7_Templates := "value_type := Int" } "IEC_Counter_0_DB 10".CTU(r := "Potlife".contol."reset counter", pv := 60, cv => "Potlife"."Time PV"."secPulse PV")
      Coil( "Potlife".contol."60sec pulse done" )
   END_RUNG
   // the same network as SCL:
   #_w1 := "Potlife".contol."start potlife timer" AND "Potlife"."potlife time in minutes";
   "IEC_Timer_0_DB_2".TON(IN := #_w1,
                          PT := "Potlife"."set time input".minutes,
                          ET => "Potlife"."Time PV".minutestimerPV);
   "Potlife".contol."minutes timer Done" := "IEC_Timer_0_DB_2".Q;
   "IEC_Counter_0_DB 10".CTU(CU := #_w1 AND NOT "Potlife".contol."minutes timer Done" AND "Clock_1Hz",
                           R := "Potlife".contol."reset counter",
                           PV := 60,
                           CV => "Potlife"."Time PV"."secPulse PV");
   "Potlife".contol."60sec pulse done" := "IEC_Counter_0_DB 10".Q;
END_REGION

REGION Network 9: Potlife Elapsed
   RUNG wire#powerrail
      Contact( "Potlife".contol."Seconds timer Done" )
      wire#w1
      S_Coil( "Potlife".contol."Potlife elapsed Start Regeneration" )
   END_RUNG
   RUNG wire#powerrail
      Contact( "Potlife".contol."minutes timer Done" )
   END_RUNG wire#w1
   // the same network as SCL:
   IF "Potlife".contol."Seconds timer Done" OR "Potlife".contol."minutes timer Done" THEN
       "Potlife".contol."Potlife elapsed Start Regeneration" := TRUE;
   END_IF;
END_REGION

REGION Network 10: reset upcount
   RUNG wire#powerrail
      Contact( "Potlife".contol."60sec pulse done" )
      wire#w1
      Coil( "Potlife".contol."reset counter" )
   END_RUNG
   RUNG wire#powerrail
      Contact( "Potlife".contol."Potlife elapsed Start Regeneration" )
   END_RUNG wire#w1
   RUNG wire#powerrail
      Contact( "Potlife".contol."minutes timer Done" )
   END_RUNG wire#w1
   RUNG wire#powerrail
      I_Contact( "Potlife".contol."start potlife timer" )
   END_RUNG wire#w1
   // the same network as SCL:
   "Potlife".contol."reset counter" := "Potlife".contol."60sec pulse done" OR "Potlife".contol."Potlife elapsed Start Regeneration" OR "Potlife".contol."minutes timer Done" OR NOT "Potlife".contol."start potlife timer";
END_REGION

REGION Network 11: Timer PV not scalled
   RUNG wire#powerrail
      Div(in1 := "Potlife"."Time PV"."Sectimer PV", in2 := 1000, out => "Potlife"."Time PV unscalled"."Sectimer PV")
      Div(in1 := "Potlife"."Time PV".minutestimerPV, in2 := 60000, out => "Potlife"."Time PV unscalled".minutestimerPV)
   END_RUNG
   // the same network as SCL:
   "Potlife"."Time PV unscalled"."Sectimer PV" := "Potlife"."Time PV"."Sectimer PV" / 1000;
   "Potlife"."Time PV unscalled".minutestimerPV := "Potlife"."Time PV".minutestimerPV / 60000;
END_REGION

REGION Network 12: run time down count
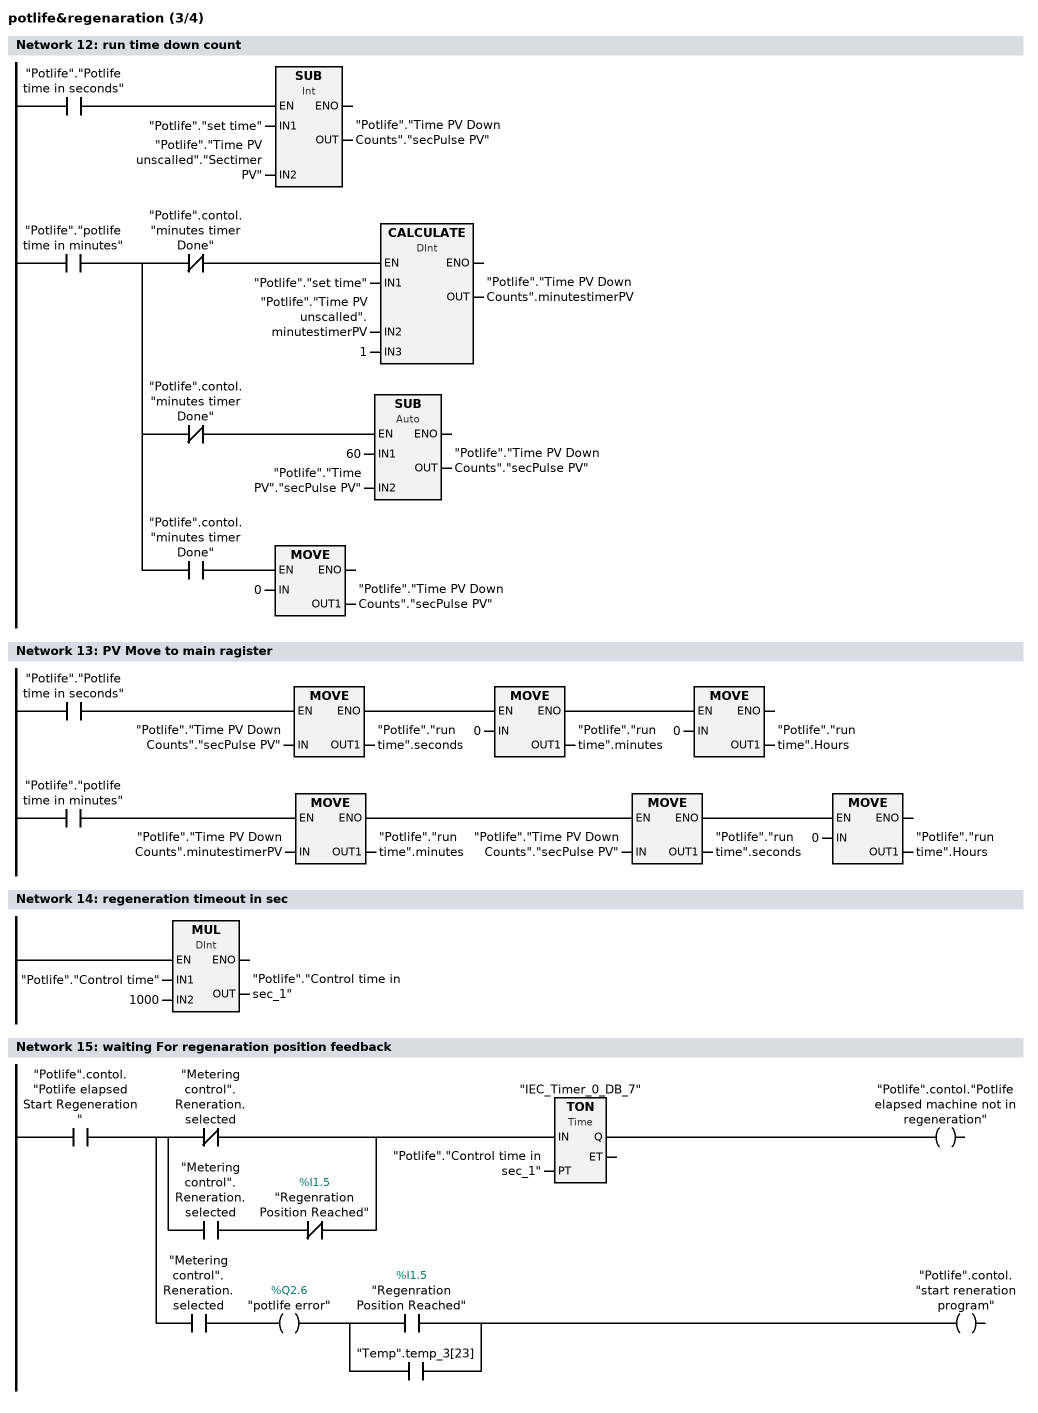
   RUNG wire#powerrail
      Contact( "Potlife"."Potlife time in seconds" )
      { S7_Templates := "SrcType := Int" } Sub(in1 := "Potlife"."set time", in2 := "Potlife"."Time PV unscalled"."Sectimer PV", out => "Potlife"."Time PV Down Counts"."secPulse PV")
   END_RUNG
   RUNG wire#powerrail
      Contact( "Potlife"."potlife time in minutes" )
      wire#w1
      I_Contact( "Potlife".contol."minutes timer Done" )
      { S7_Templates := "SrcType := DInt"; S7_Expression := "IN1-IN2-IN3" } Calculate(in1 := "Potlife"."set time", in2 := "Potlife"."Time PV unscalled".minutestimerPV, in3 := 1, out => "Potlife"."Time PV Down Counts".minutestimerPV)
   END_RUNG
   RUNG wire#w1
      I_Contact( "Potlife".contol."minutes timer Done" )
      Sub(in1 := 60, in2 := "Potlife"."Time PV"."secPulse PV", out => "Potlife"."Time PV Down Counts"."secPulse PV")
   END_RUNG
   RUNG wire#w1
      Contact( "Potlife".contol."minutes timer Done" )
      Move(in := 0, out1 => "Potlife"."Time PV Down Counts"."secPulse PV")
   END_RUNG
   // the same network as SCL:
   IF "Potlife"."Potlife time in seconds" THEN
       "Potlife"."Time PV Down Counts"."secPulse PV" := "Potlife"."set time" - "Potlife"."Time PV unscalled"."Sectimer PV";
   END_IF;
   IF "Potlife"."potlife time in minutes" AND NOT "Potlife".contol."minutes timer Done" THEN
       "Potlife"."Time PV Down Counts".minutestimerPV := "Potlife"."set time"-"Potlife"."Time PV unscalled".minutestimerPV-1;
       "Potlife"."Time PV Down Counts"."secPulse PV" := 60 - "Potlife"."Time PV"."secPulse PV";
   END_IF;
   IF "Potlife"."potlife time in minutes" AND "Potlife".contol."minutes timer Done" THEN
       "Potlife"."Time PV Down Counts"."secPulse PV" := 0;
   END_IF;
END_REGION

REGION Network 13: PV Move to main ragister
   RUNG wire#powerrail
      Contact( "Potlife"."Potlife time in seconds" )
      Move(in := "Potlife"."Time PV Down Counts"."secPulse PV", out1 => "Potlife"."run time".seconds)
      Move(in := 0, out1 => "Potlife"."run time".minutes)
      Move(in := 0, out1 => "Potlife"."run time".Hours)
   END_RUNG
   RUNG wire#powerrail
      Contact( "Potlife"."potlife time in minutes" )
      Move(in := "Potlife"."Time PV Down Counts".minutestimerPV, out1 => "Potlife"."run time".minutes)
      Move(in := "Potlife"."Time PV Down Counts"."secPulse PV", out1 => "Potlife"."run time".seconds)
      Move(in := 0, out1 => "Potlife"."run time".Hours)
   END_RUNG
   // the same network as SCL:
   IF "Potlife"."Potlife time in seconds" THEN
       "Potlife"."run time".seconds := "Potlife"."Time PV Down Counts"."secPulse PV";
       "Potlife"."run time".minutes := 0;
       "Potlife"."run time".Hours := 0;
   END_IF;
   IF "Potlife"."potlife time in minutes" THEN
       "Potlife"."run time".minutes := "Potlife"."Time PV Down Counts".minutestimerPV;
       "Potlife"."run time".seconds := "Potlife"."Time PV Down Counts"."secPulse PV";
       "Potlife"."run time".Hours := 0;
   END_IF;
END_REGION

REGION Network 14: regeneration timeout in sec
   RUNG wire#powerrail
      { S7_Templates := "SrcType := DInt" } Mul(in1 := "Potlife"."Control time", in2 := 1000, out => "Potlife"."Control time in sec_1")
   END_RUNG
   // the same network as SCL:
   "Potlife"."Control time in sec_1" := "Potlife"."Control time" * 1000;
END_REGION

REGION Network 15: waiting For regenaration position feedback
   RUNG wire#powerrail
      Contact( "Potlife".contol."Potlife elapsed Start Regeneration" )
      wire#w1
      I_Contact( "Metering control".Reneration.selected )
      wire#w2
      { S7_Templates := "time_type := Time" } "IEC_Timer_0_DB_7".TON(pt := "Potlife"."Control time in sec_1", et =>)
      Coil( "Potlife".contol."Potlife elapsed machine not in regeneration" )
   END_RUNG
   RUNG wire#w1
      Contact( "Metering control".Reneration.selected )
      I_Contact( "Regenration Position Reached" )
   END_RUNG wire#w2
   RUNG wire#w1
      Contact( "Metering control".Reneration.selected )
      Coil( "potlife error" )
      wire#w3
      Contact( "Regenration Position Reached" )
      wire#w4
      Coil( "Potlife".contol."start reneration program" )
   END_RUNG
   RUNG wire#w3
      Contact( "Temp".temp_3[23] )
   END_RUNG wire#w4
   // the same network as SCL:
   "IEC_Timer_0_DB_7".TON(IN := "Potlife".contol."Potlife elapsed Start Regeneration" AND (NOT "Metering control".Reneration.selected OR ("Metering control".Reneration.selected AND NOT "Regenration Position Reached")),
                          PT := "Potlife"."Control time in sec_1");
   "Potlife".contol."Potlife elapsed machine not in regeneration" := "IEC_Timer_0_DB_7".Q;
   "potlife error" := "Potlife".contol."Potlife elapsed Start Regeneration" AND "Metering control".Reneration.selected;
   "Potlife".contol."start reneration program" := "potlife error" AND ("Regenration Position Reached" OR "Temp".temp_3[23]);
END_REGION

REGION Network 16: Selecting regeneration program
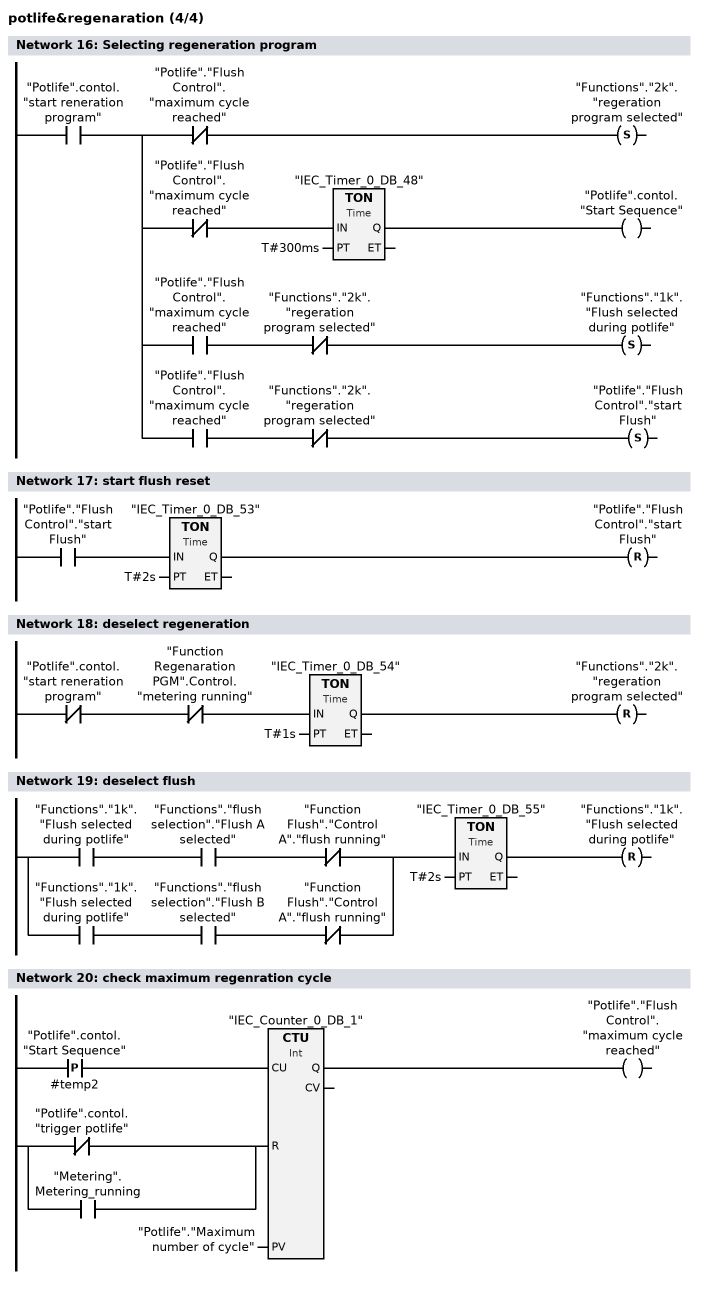
   RUNG wire#powerrail
      Contact( "Potlife".contol."start reneration program" )
      wire#w1
      I_Contact( "Potlife"."Flush Control"."maximum cycle reached" )
      S_Coil( "Functions"."2k"."regeration program selected" )
   END_RUNG
   RUNG wire#w1
      I_Contact( "Potlife"."Flush Control"."maximum cycle reached" )
      { S7_Templates := "time_type := Time" } "IEC_Timer_0_DB_48".TON(pt := T#300ms, et =>)
      Coil( "Potlife".contol."Start Sequence" )
   END_RUNG
   RUNG wire#w1
      Contact( "Potlife"."Flush Control"."maximum cycle reached" )
      I_Contact( "Functions"."2k"."regeration program selected" )
      S_Coil( "Functions"."1k"."Flush selected during potlife" )
   END_RUNG
   RUNG wire#w1
      Contact( "Potlife"."Flush Control"."maximum cycle reached" )
      I_Contact( "Functions"."2k"."regeration program selected" )
      S_Coil( "Potlife"."Flush Control"."start Flush" )
   END_RUNG
   // the same network as SCL:
   IF "Potlife".contol."start reneration program" AND NOT "Potlife"."Flush Control"."maximum cycle reached" THEN
       "Functions"."2k"."regeration program selected" := TRUE;
   END_IF;
   "IEC_Timer_0_DB_48".TON(IN := "Potlife".contol."start reneration program" AND NOT "Potlife"."Flush Control"."maximum cycle reached",
                           PT := T#300ms);
   "Potlife".contol."Start Sequence" := "IEC_Timer_0_DB_48".Q;
   IF "Potlife".contol."start reneration program" AND "Potlife"."Flush Control"."maximum cycle reached" AND NOT "Functions"."2k"."regeration program selected" THEN
       "Functions"."1k"."Flush selected during potlife" := TRUE;
       "Potlife"."Flush Control"."start Flush" := TRUE;
   END_IF;
END_REGION

REGION Network 17: start flush reset
   RUNG wire#powerrail
      Contact( "Potlife"."Flush Control"."start Flush" )
      { S7_Templates := "time_type := Time" } "IEC_Timer_0_DB_53".TON(pt := T#2s, et =>)
      R_Coil( "Potlife"."Flush Control"."start Flush" )
   END_RUNG
   // the same network as SCL:
   "IEC_Timer_0_DB_53".TON(IN := "Potlife"."Flush Control"."start Flush", PT := T#2s);
   IF "IEC_Timer_0_DB_53".Q THEN "Potlife"."Flush Control"."start Flush" := FALSE; END_IF;
END_REGION

REGION Network 18: deselect regeneration
   RUNG wire#powerrail
      I_Contact( "Potlife".contol."start reneration program" )
      I_Contact( "Function Regenaration PGM".Control."metering running" )
      { S7_Templates := "time_type := Time" } "IEC_Timer_0_DB_54".TON(pt := T#1s, et =>)
      R_Coil( "Functions"."2k"."regeration program selected" )
   END_RUNG
   // the same network as SCL:
   "IEC_Timer_0_DB_54".TON(IN := NOT "Potlife".contol."start reneration program" AND NOT "Function Regenaration PGM".Control."metering running",
                           PT := T#1s);
   IF "IEC_Timer_0_DB_54".Q THEN "Functions"."2k"."regeration program selected" := FALSE; END_IF;
END_REGION

REGION Network 19: deselect flush
   RUNG wire#powerrail
      Contact( "Functions"."1k"."Flush selected during potlife" )
      Contact( "Functions"."flush selection"."Flush A selected" )
      I_Contact( "Function Flush"."Control A"."flush running" )
      wire#w1
      { S7_Templates := "time_type := Time" } "IEC_Timer_0_DB_55".TON(pt := T#2s, et =>)
      R_Coil( "Functions"."1k"."Flush selected during potlife" )
   END_RUNG
   RUNG wire#powerrail
      Contact( "Functions"."1k"."Flush selected during potlife" )
      Contact( "Functions"."flush selection"."Flush B selected" )
      I_Contact( "Function Flush"."Control A"."flush running" )
   END_RUNG wire#w1
   // the same network as SCL:
   "IEC_Timer_0_DB_55".TON(IN := ("Functions"."1k"."Flush selected during potlife" AND "Functions"."flush selection"."Flush A selected" AND NOT "Function Flush"."Control A"."flush running") OR ("Functions"."1k"."Flush selected during potlife" AND "Functions"."flush selection"."Flush B selected" AND NOT "Function Flush"."Control A"."flush running"),
                           PT := T#2s);
   IF "IEC_Timer_0_DB_55".Q THEN "Functions"."1k"."Flush selected during potlife" := FALSE; END_IF;
END_REGION

REGION Network 20: check maximum regenration cycle
   RUNG wire#powerrail
      P_Contact(operand := "Potlife".contol."Start Sequence", bit := #temp2)
      { S7_Templates := "value_type := Int" } "IEC_Counter_0_DB_1".CTU(r := wire#w1, pv := "Potlife"."Maximum number of cycle", cv =>)
      Coil( "Potlife"."Flush Control"."maximum cycle reached" )
   END_RUNG
   RUNG wire#powerrail
      I_Contact( "Potlife".contol."trigger potlife" )
   END_RUNG wire#w1
   RUNG wire#powerrail
      Contact( "Metering".Metering_running )
   END_RUNG wire#w1
   // the same network as SCL:
   #_w1 := "Potlife".contol."Start Sequence" AND NOT #temp2;   // rising edge of "Potlife".contol."Start Sequence"
   #temp2 := "Potlife".contol."Start Sequence";
   "IEC_Counter_0_DB_1".CTU(CU := #_w1,
                           R := NOT "Potlife".contol."trigger potlife" OR "Metering".Metering_running,
                           PV := "Potlife"."Maximum number of cycle");
   "Potlife"."Flush Control"."maximum cycle reached" := "IEC_Counter_0_DB_1".Q;
END_REGION
END_FUNCTION

FUNCTION "level Control" : Void   // FC20, LAD
{ S7_Optimized_Access := 'TRUE' }
VERSION : 0.1
// stored: AutoNumber true, IsIECCheckEnabled false, SetENOAutomatically false, UDAEnableTagReadback false
   VAR_TEMP   // added for the SCL form of the ladder/FBD networks
      _w1 : Bool;
   END_VAR
BEGIN

REGION Network 1: Level Sensor Tank A
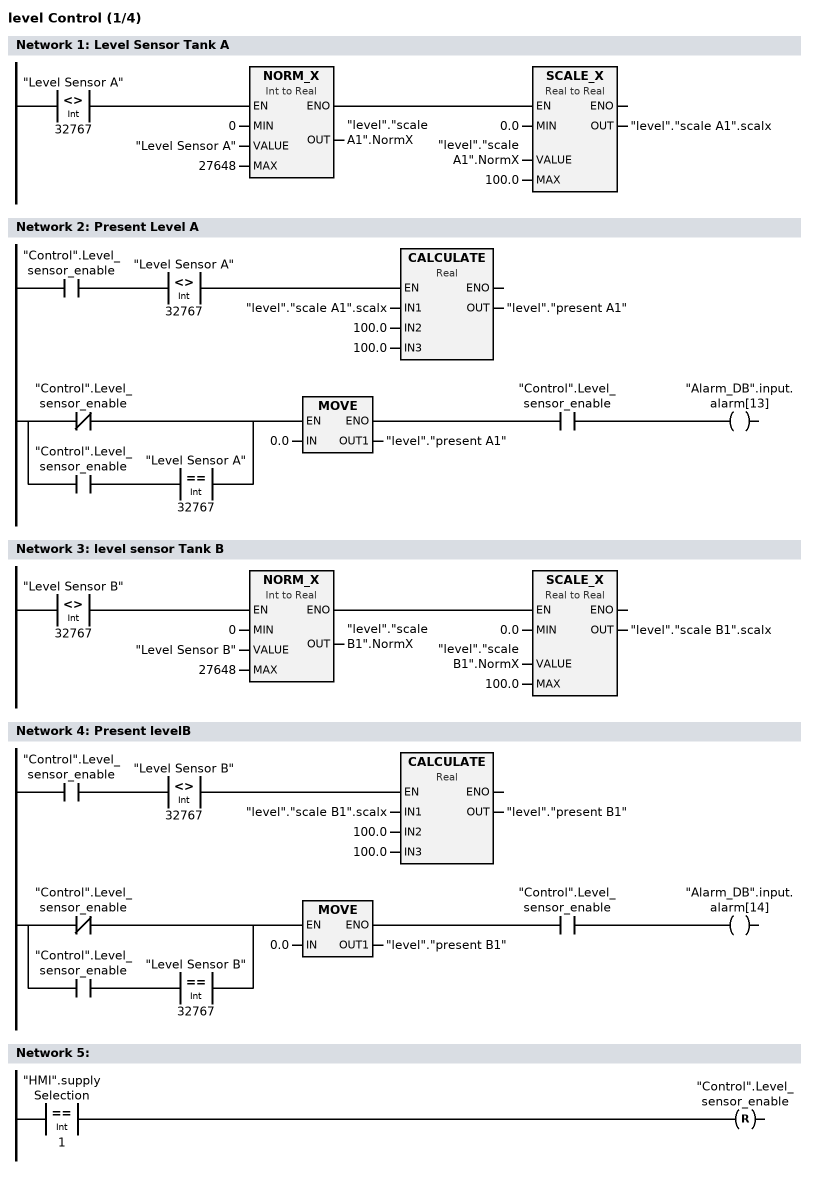
   RUNG wire#powerrail
      { S7_Templates := "SrcType := Int" } NE_Contact(in1 := "Level Sensor A", in2 := 32767)
      { S7_Templates := "[SrcType := Int, DestType := Real]" } Normalize(min := 0, value := "Level Sensor A", max := 27648, out => "level"."scale A1".NormX)
      { S7_Templates := "[SrcType := Real, DestType := Real]" } Scale(min := 0.0, value := "level"."scale A1".NormX, max := 100.0, out => "level"."scale A1".scalx)
   END_RUNG
   // the same network as SCL:
   IF "Level Sensor A" <> 32767 THEN
       "level"."scale A1".NormX := NORM_X(MIN := 0, VALUE := "Level Sensor A", MAX := 27648);
       "level"."scale A1".scalx := SCALE_X(MIN := 0.0, VALUE := "level"."scale A1".NormX, MAX := 100.0);
   END_IF;
END_REGION

REGION Network 2: Present Level A
   RUNG wire#powerrail
      Contact( "Control".Level_sensor_enable )
      { S7_Templates := "SrcType := Int" } NE_Contact(in1 := "Level Sensor A", in2 := 32767)
      { S7_Templates := "SrcType := Real"; S7_Expression := "ROUND(IN1*IN2)/IN3" } Calculate(in1 := "level"."scale A1".scalx, in2 := 100.0, in3 := 100.0, out => "level"."present A1")
   END_RUNG
   RUNG wire#powerrail
      I_Contact( "Control".Level_sensor_enable )
      wire#w1
      Move(in := 0.0, out1 => "level"."present A1")
      Contact( "Control".Level_sensor_enable )
      Coil( "Alarm_DB".input.alarm[13] )
   END_RUNG
   RUNG wire#powerrail
      Contact( "Control".Level_sensor_enable )
      { S7_Templates := "SrcType := Int" } EQ_Contact(in1 := "Level Sensor A", in2 := 32767)
   END_RUNG wire#w1
   // the same network as SCL:
   IF "Control".Level_sensor_enable AND ("Level Sensor A" <> 32767) THEN
       "level"."present A1" := ROUND("level"."scale A1".scalx*100.0)/100.0;
   END_IF;
   #_w1 := NOT "Control".Level_sensor_enable OR ("Control".Level_sensor_enable AND ("Level Sensor A" = 32767));
   IF #_w1 THEN "level"."present A1" := 0.0; END_IF;
   "Alarm_DB".input.alarm[13] := #_w1 AND "Control".Level_sensor_enable;
END_REGION

REGION Network 3: level sensor Tank B
   RUNG wire#powerrail
      { S7_Templates := "SrcType := Int" } NE_Contact(in1 := "Level Sensor B", in2 := 32767)
      { S7_Templates := "[SrcType := Int, DestType := Real]" } Normalize(min := 0, value := "Level Sensor B", max := 27648, out => "level"."scale B1".NormX)
      { S7_Templates := "[SrcType := Real, DestType := Real]" } Scale(min := 0.0, value := "level"."scale B1".NormX, max := 100.0, out => "level"."scale B1".scalx)
   END_RUNG
   // the same network as SCL:
   IF "Level Sensor B" <> 32767 THEN
       "level"."scale B1".NormX := NORM_X(MIN := 0, VALUE := "Level Sensor B", MAX := 27648);
       "level"."scale B1".scalx := SCALE_X(MIN := 0.0, VALUE := "level"."scale B1".NormX, MAX := 100.0);
   END_IF;
END_REGION

REGION Network 4: Present levelB
   RUNG wire#powerrail
      Contact( "Control".Level_sensor_enable )
      { S7_Templates := "SrcType := Int" } NE_Contact(in1 := "Level Sensor B", in2 := 32767)
      { S7_Templates := "SrcType := Real"; S7_Expression := "ROUND(IN1*IN2)/IN3" } Calculate(in1 := "level"."scale B1".scalx, in2 := 100.0, in3 := 100.0, out => "level"."present B1")
   END_RUNG
   RUNG wire#powerrail
      I_Contact( "Control".Level_sensor_enable )
      wire#w1
      Move(in := 0.0, out1 => "level"."present B1")
      Contact( "Control".Level_sensor_enable )
      Coil( "Alarm_DB".input.alarm[14] )
   END_RUNG
   RUNG wire#powerrail
      Contact( "Control".Level_sensor_enable )
      { S7_Templates := "SrcType := Int" } EQ_Contact(in1 := "Level Sensor B", in2 := 32767)
   END_RUNG wire#w1
   // the same network as SCL:
   IF "Control".Level_sensor_enable AND ("Level Sensor B" <> 32767) THEN
       "level"."present B1" := ROUND("level"."scale B1".scalx*100.0)/100.0;
   END_IF;
   #_w1 := NOT "Control".Level_sensor_enable OR ("Control".Level_sensor_enable AND ("Level Sensor B" = 32767));
   IF #_w1 THEN "level"."present B1" := 0.0; END_IF;
   "Alarm_DB".input.alarm[14] := #_w1 AND "Control".Level_sensor_enable;
END_REGION

REGION Network 5
   RUNG wire#powerrail
      { S7_Templates := "SrcType := Int" } EQ_Contact(in1 := "HMI".supplySelection, in2 := 1)
      R_Coil( "Control".Level_sensor_enable )
   END_RUNG
   // the same network as SCL:
   IF "HMI".supplySelection = 1 THEN "Control".Level_sensor_enable := FALSE; END_IF;
END_REGION

REGION Network 6: Low level A
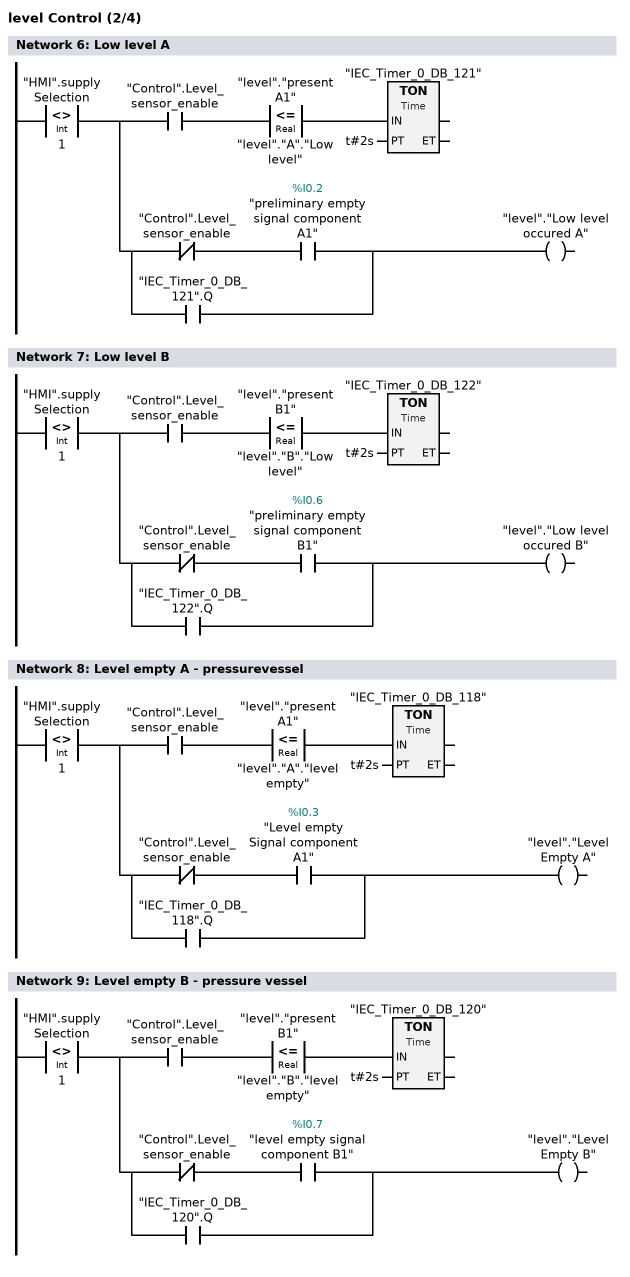
   RUNG wire#powerrail
      { S7_Templates := "SrcType := Int" } NE_Contact(in1 := "HMI".supplySelection, in2 := 1)
      wire#w1
      Contact( "Control".Level_sensor_enable )
      { S7_Templates := "SrcType := Real" } LE_Contact(in1 := "level"."present A1", in2 := "level"."A"."Low level")
      { S7_Templates := "time_type := Time" } "IEC_Timer_0_DB_121".TON(pt := t#2s, et =>)
   END_RUNG
   RUNG wire#w1
      I_Contact( "Control".Level_sensor_enable )
      Contact( "preliminary empty signal component A1" )
      wire#w2
      Coil( "level"."Low level occured A" )
   END_RUNG
   RUNG wire#w1
      Contact( "IEC_Timer_0_DB_121".Q )
   END_RUNG wire#w2
   // the same network as SCL:
   #_w1 := "HMI".supplySelection <> 1;
   "IEC_Timer_0_DB_121".TON(IN := #_w1 AND "Control".Level_sensor_enable AND ("level"."present A1" <= "level"."A"."Low level"),
                           PT := t#2s);
   "level"."Low level occured A" := #_w1 AND ((NOT "Control".Level_sensor_enable AND "preliminary empty signal component A1") OR "IEC_Timer_0_DB_121".Q);
END_REGION

REGION Network 7: Low level B
   RUNG wire#powerrail
      { S7_Templates := "SrcType := Int" } NE_Contact(in1 := "HMI".supplySelection, in2 := 1)
      wire#w1
      Contact( "Control".Level_sensor_enable )
      { S7_Templates := "SrcType := Real" } LE_Contact(in1 := "level"."present B1", in2 := "level"."B"."Low level")
      { S7_Templates := "time_type := Time" } "IEC_Timer_0_DB_122".TON(pt := t#2s, et =>)
   END_RUNG
   RUNG wire#w1
      I_Contact( "Control".Level_sensor_enable )
      Contact( "preliminary empty signal component B1" )
      wire#w2
      Coil( "level"."Low level occured B" )
   END_RUNG
   RUNG wire#w1
      Contact( "IEC_Timer_0_DB_122".Q )
   END_RUNG wire#w2
   // the same network as SCL:
   #_w1 := "HMI".supplySelection <> 1;
   "IEC_Timer_0_DB_122".TON(IN := #_w1 AND "Control".Level_sensor_enable AND ("level"."present B1" <= "level"."B"."Low level"),
                           PT := t#2s);
   "level"."Low level occured B" := #_w1 AND ((NOT "Control".Level_sensor_enable AND "preliminary empty signal component B1") OR "IEC_Timer_0_DB_122".Q);
END_REGION

REGION Network 8: Level empty A - pressurevessel
   RUNG wire#powerrail
      { S7_Templates := "SrcType := Int" } NE_Contact(in1 := "HMI".supplySelection, in2 := 1)
      wire#w1
      Contact( "Control".Level_sensor_enable )
      { S7_Templates := "SrcType := Real" } LE_Contact(in1 := "level"."present A1", in2 := "level"."A"."level empty")
      { S7_Templates := "time_type := Time" } "IEC_Timer_0_DB_118".TON(pt := t#2s, et =>)
   END_RUNG
   RUNG wire#w1
      I_Contact( "Control".Level_sensor_enable )
      Contact( "Level empty Signal component A1" )
      wire#w2
      Coil( "level"."Level Empty A" )
   END_RUNG
   RUNG wire#w1
      Contact( "IEC_Timer_0_DB_118".Q )
   END_RUNG wire#w2
   // the same network as SCL:
   #_w1 := "HMI".supplySelection <> 1;
   "IEC_Timer_0_DB_118".TON(IN := #_w1 AND "Control".Level_sensor_enable AND ("level"."present A1" <= "level"."A"."level empty"),
                           PT := t#2s);
   "level"."Level Empty A" := #_w1 AND ((NOT "Control".Level_sensor_enable AND "Level empty Signal component A1") OR "IEC_Timer_0_DB_118".Q);
END_REGION

REGION Network 9: Level empty B - pressure vessel
   RUNG wire#powerrail
      { S7_Templates := "SrcType := Int" } NE_Contact(in1 := "HMI".supplySelection, in2 := 1)
      wire#w1
      Contact( "Control".Level_sensor_enable )
      { S7_Templates := "SrcType := Real" } LE_Contact(in1 := "level"."present B1", in2 := "level"."B"."level empty")
      { S7_Templates := "time_type := Time" } "IEC_Timer_0_DB_120".TON(pt := t#2s, et =>)
   END_RUNG
   RUNG wire#w1
      I_Contact( "Control".Level_sensor_enable )
      Contact( "level empty signal component B1" )
      wire#w2
      Coil( "level"."Level Empty B" )
   END_RUNG
   RUNG wire#w1
      Contact( "IEC_Timer_0_DB_120".Q )
   END_RUNG wire#w2
   // the same network as SCL:
   #_w1 := "HMI".supplySelection <> 1;
   "IEC_Timer_0_DB_120".TON(IN := #_w1 AND "Control".Level_sensor_enable AND ("level"."present B1" <= "level"."B"."level empty"),
                           PT := t#2s);
   "level"."Level Empty B" := #_w1 AND ((NOT "Control".Level_sensor_enable AND "level empty signal component B1") OR "IEC_Timer_0_DB_120".Q);
END_REGION

REGION Network 10: High Level A - Pressure vessel
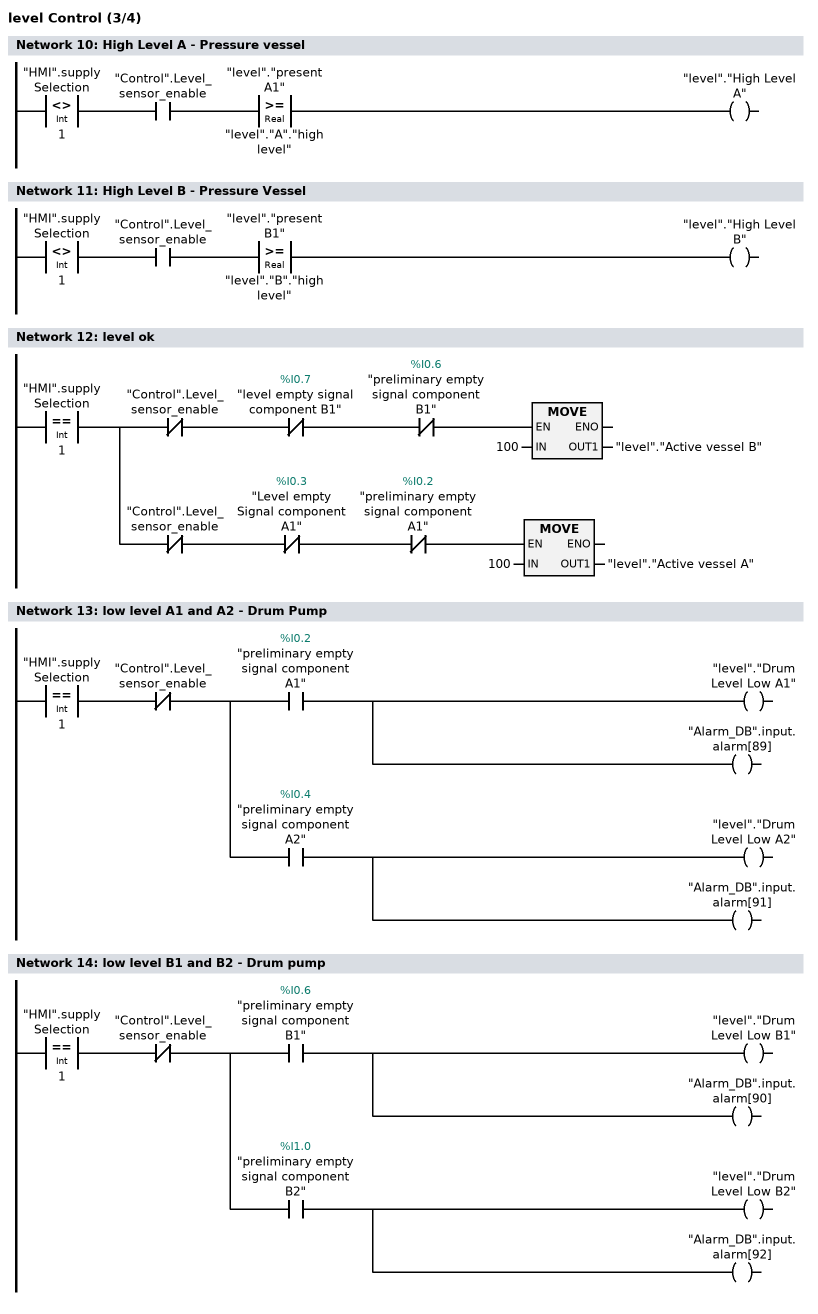
   RUNG wire#powerrail
      { S7_Templates := "SrcType := Int" } NE_Contact(in1 := "HMI".supplySelection, in2 := 1)
      Contact( "Control".Level_sensor_enable )
      { S7_Templates := "SrcType := Real" } GE_Contact(in1 := "level"."present A1", in2 := "level"."A"."high level")
      Coil( "level"."High Level A" )
   END_RUNG
   // the same network as SCL:
   "level"."High Level A" := ("HMI".supplySelection <> 1) AND "Control".Level_sensor_enable AND ("level"."present A1" >= "level"."A"."high level");
END_REGION

REGION Network 11: High Level B - Pressure Vessel
   RUNG wire#powerrail
      { S7_Templates := "SrcType := Int" } NE_Contact(in1 := "HMI".supplySelection, in2 := 1)
      Contact( "Control".Level_sensor_enable )
      { S7_Templates := "SrcType := Real" } GE_Contact(in1 := "level"."present B1", in2 := "level"."B"."high level")
      Coil( "level"."High Level B" )
   END_RUNG
   // the same network as SCL:
   "level"."High Level B" := ("HMI".supplySelection <> 1) AND "Control".Level_sensor_enable AND ("level"."present B1" >= "level"."B"."high level");
END_REGION

REGION Network 12: level ok
   RUNG wire#powerrail
      { S7_Templates := "SrcType := Int" } EQ_Contact(in1 := "HMI".supplySelection, in2 := 1)
      wire#w1
      I_Contact( "Control".Level_sensor_enable )
      I_Contact( "level empty signal component B1" )
      I_Contact( "preliminary empty signal component B1" )
      Move(in := 100, out1 => "level"."Active vessel B")
   END_RUNG
   RUNG wire#w1
      I_Contact( "Control".Level_sensor_enable )
      I_Contact( "Level empty Signal component A1" )
      I_Contact( "preliminary empty signal component A1" )
      Move(in := 100, out1 => "level"."Active vessel A")
   END_RUNG
   // the same network as SCL:
   #_w1 := "HMI".supplySelection = 1;
   IF #_w1 AND NOT "Control".Level_sensor_enable AND NOT "level empty signal component B1" AND NOT "preliminary empty signal component B1" THEN
       "level"."Active vessel B" := 100;
   END_IF;
   IF #_w1 AND NOT "Control".Level_sensor_enable AND NOT "Level empty Signal component A1" AND NOT "preliminary empty signal component A1" THEN
       "level"."Active vessel A" := 100;
   END_IF;
END_REGION

REGION Network 13: low level A1 and A2 - Drum Pump
   RUNG wire#powerrail
      { S7_Templates := "SrcType := Int" } EQ_Contact(in1 := "HMI".supplySelection, in2 := 1)
      I_Contact( "Control".Level_sensor_enable )
      wire#w1
      Contact( "preliminary empty signal component A1" )
      wire#w2
      Coil( "level"."Drum Level Low A1" )
   END_RUNG
   RUNG wire#w2
      Coil( "Alarm_DB".input.alarm[89] )
   END_RUNG
   RUNG wire#w1
      Contact( "preliminary empty signal component A2" )
      wire#w3
      Coil( "level"."Drum Level Low A2" )
   END_RUNG
   RUNG wire#w3
      Coil( "Alarm_DB".input.alarm[91] )
   END_RUNG
   // the same network as SCL:
   #_w1 := ("HMI".supplySelection = 1) AND NOT "Control".Level_sensor_enable;
   "level"."Drum Level Low A1" := #_w1 AND "preliminary empty signal component A1";
   "Alarm_DB".input.alarm[89] := "level"."Drum Level Low A1";
   "level"."Drum Level Low A2" := #_w1 AND "preliminary empty signal component A2";
   "Alarm_DB".input.alarm[91] := "level"."Drum Level Low A2";
END_REGION

REGION Network 14: low level B1 and B2 - Drum pump
   RUNG wire#powerrail
      { S7_Templates := "SrcType := Int" } EQ_Contact(in1 := "HMI".supplySelection, in2 := 1)
      I_Contact( "Control".Level_sensor_enable )
      wire#w1
      Contact( "preliminary empty signal component B1" )
      wire#w2
      Coil( "level"."Drum Level Low B1" )
   END_RUNG
   RUNG wire#w2
      Coil( "Alarm_DB".input.alarm[90] )
   END_RUNG
   RUNG wire#w1
      Contact( "preliminary empty signal component B2" )
      wire#w3
      Coil( "level"."Drum Level Low B2" )
   END_RUNG
   RUNG wire#w3
      Coil( "Alarm_DB".input.alarm[92] )
   END_RUNG
   // the same network as SCL:
   #_w1 := ("HMI".supplySelection = 1) AND NOT "Control".Level_sensor_enable;
   "level"."Drum Level Low B1" := #_w1 AND "preliminary empty signal component B1";
   "Alarm_DB".input.alarm[90] := "level"."Drum Level Low B1";
   "level"."Drum Level Low B2" := #_w1 AND "preliminary empty signal component B2";
   "Alarm_DB".input.alarm[92] := "level"."Drum Level Low B2";
END_REGION

REGION Network 15: level empty A1 and A2 - Drum pump
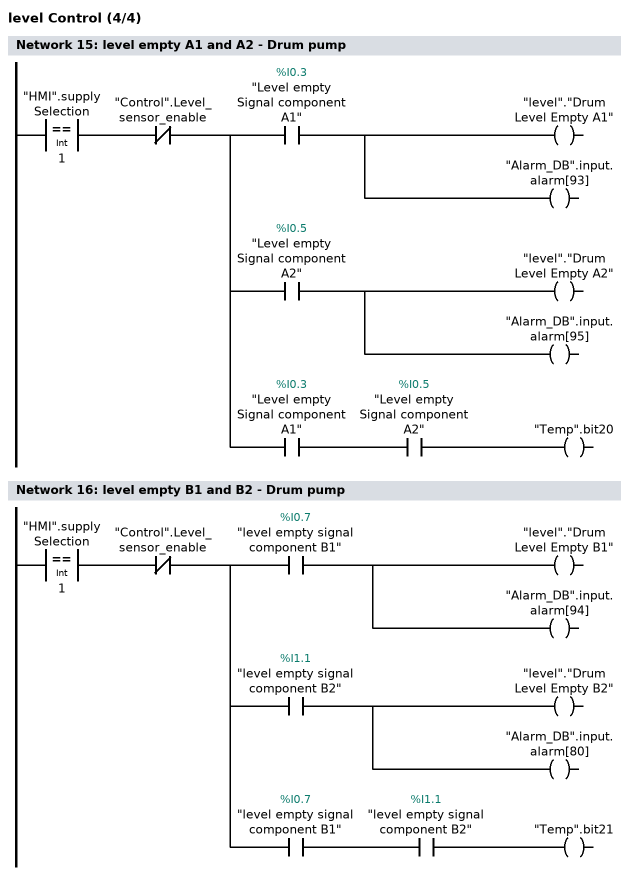
   RUNG wire#powerrail
      { S7_Templates := "SrcType := Int" } EQ_Contact(in1 := "HMI".supplySelection, in2 := 1)
      I_Contact( "Control".Level_sensor_enable )
      wire#w1
      Contact( "Level empty Signal component A1" )
      wire#w2
      Coil( "level"."Drum Level Empty A1" )
   END_RUNG
   RUNG wire#w2
      Coil( "Alarm_DB".input.alarm[93] )
   END_RUNG
   RUNG wire#w1
      Contact( "Level empty Signal component A2" )
      wire#w3
      Coil( "level"."Drum Level Empty A2" )
   END_RUNG
   RUNG wire#w3
      Coil( "Alarm_DB".input.alarm[95] )
   END_RUNG
   RUNG wire#w1
      Contact( "Level empty Signal component A1" )
      Contact( "Level empty Signal component A2" )
      Coil( "Temp".bit20 )
   END_RUNG
   // the same network as SCL:
   #_w1 := ("HMI".supplySelection = 1) AND NOT "Control".Level_sensor_enable;
   "level"."Drum Level Empty A1" := #_w1 AND "Level empty Signal component A1";
   "Alarm_DB".input.alarm[93] := "level"."Drum Level Empty A1";
   "level"."Drum Level Empty A2" := #_w1 AND "Level empty Signal component A2";
   "Alarm_DB".input.alarm[95] := "level"."Drum Level Empty A2";
   "Temp".bit20 := #_w1 AND "Level empty Signal component A1" AND "Level empty Signal component A2";
END_REGION

REGION Network 16: level empty B1 and B2 - Drum pump
   RUNG wire#powerrail
      { S7_Templates := "SrcType := Int" } EQ_Contact(in1 := "HMI".supplySelection, in2 := 1)
      I_Contact( "Control".Level_sensor_enable )
      wire#w1
      Contact( "level empty signal component B1" )
      wire#w2
      Coil( "level"."Drum Level Empty B1" )
   END_RUNG
   RUNG wire#w2
      Coil( "Alarm_DB".input.alarm[94] )
   END_RUNG
   RUNG wire#w1
      Contact( "level empty signal component B2" )
      wire#w3
      Coil( "level"."Drum Level Empty B2" )
   END_RUNG
   RUNG wire#w3
      Coil( "Alarm_DB".input.alarm[80] )
   END_RUNG
   RUNG wire#w1
      Contact( "level empty signal component B1" )
      Contact( "level empty signal component B2" )
      Coil( "Temp".bit21 )
   END_RUNG
   // the same network as SCL:
   #_w1 := ("HMI".supplySelection = 1) AND NOT "Control".Level_sensor_enable;
   "level"."Drum Level Empty B1" := #_w1 AND "level empty signal component B1";
   "Alarm_DB".input.alarm[94] := "level"."Drum Level Empty B1";
   "level"."Drum Level Empty B2" := #_w1 AND "level empty signal component B2";
   "Alarm_DB".input.alarm[80] := "level"."Drum Level Empty B2";
   "Temp".bit21 := #_w1 AND "level empty signal component B1" AND "level empty signal component B2";
END_REGION
END_FUNCTION

FUNCTION "Status" : Void   // FC27, LAD
{ S7_Optimized_Access := 'TRUE' }
VERSION : 0.1
// stored: AutoNumber true, IsIECCheckEnabled false, SetENOAutomatically false, UDAEnableTagReadback false
BEGIN

REGION Network 1: Drive control A nok
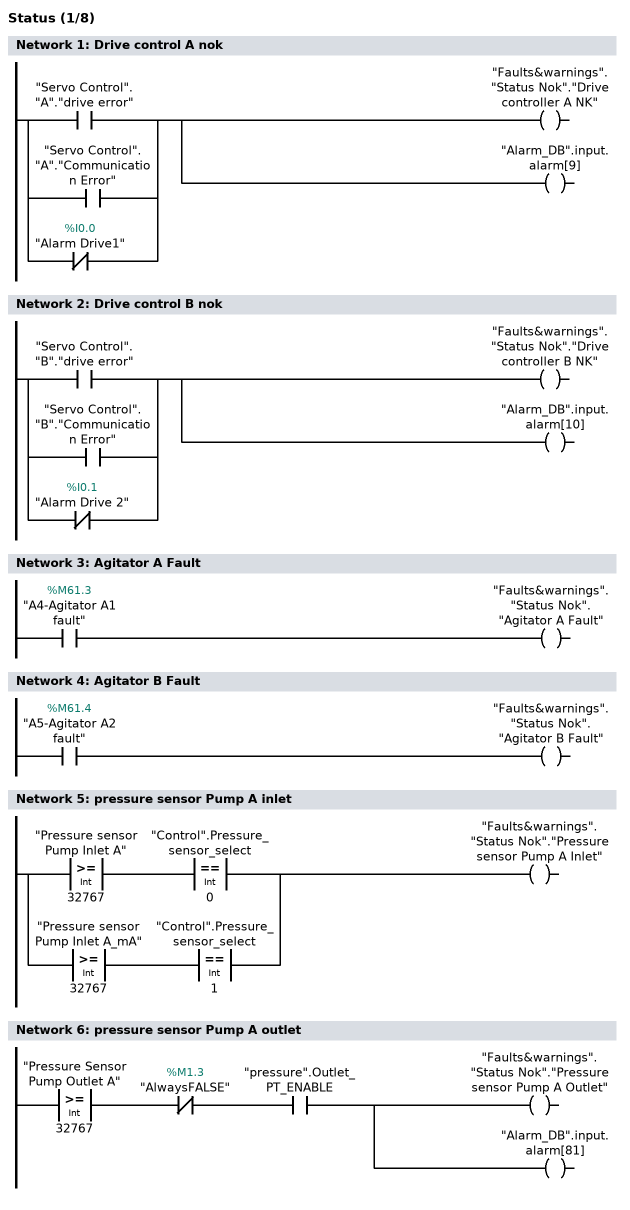
   RUNG wire#powerrail
      Contact( "Servo Control"."A"."drive error" )
      wire#w1
      Coil( "Faults&warnings"."Status Nok"."Drive controller A NK" )
   END_RUNG
   RUNG wire#powerrail
      Contact( "Servo Control"."A"."Communication Error" )
   END_RUNG wire#w1
   RUNG wire#powerrail
      I_Contact( "Alarm Drive1" )
   END_RUNG wire#w1
   RUNG wire#w1
      Coil( "Alarm_DB".input.alarm[9] )
   END_RUNG
   // the same network as SCL:
   "Faults&warnings"."Status Nok"."Drive controller A NK" := "Servo Control"."A"."drive error" OR "Servo Control"."A"."Communication Error" OR NOT "Alarm Drive1";
   "Alarm_DB".input.alarm[9] := "Faults&warnings"."Status Nok"."Drive controller A NK";
END_REGION

